# B&R Automation Studio project SD_SMA_SCADA_DEMO (part 2)

### Package Logical/SMA - SMA DataSQL demo

### GlobalDataSQL.typ - DataSQL types
```iecst
(*DataSQL types matching sma_data_collect OPC paths*)

TYPE
	DataSQLOperate_typ : 	STRUCT
		RecipeRead : BOOL;
		RecipeReadStatus : UINT;
		RecipeInsert : BOOL;
		RecipeInsertReq : BOOL;
		ProductRead : BOOL;
		ProductReadStatus : UINT;
		ProductInsert : BOOL;
		ProductInsertReq : BOOL;
		ProductInsertStatus : UDINT;
		AuditRead : BOOL;
		AuditReadStatus : UINT;
		AuditInsertFault : BOOL;
		AlarmRead : BOOL;
		AlarmReadStatus : UINT;
		AlarmInsertFault : BOOL;
		BatchInsert : BOOL;
		BatchInfoInsert : BOOL;
		RecipeCollectEnable : BOOL;
		ProductCollectEnable : BOOL;
		AlarmCollectEnable : BOOL;
		AuditCollectEnable : BOOL;
		BatchCollectEnable : BOOL;
		BatchInfoCollectEnable : BOOL;
	END_STRUCT;
END_TYPE

TYPE
	DataSQLQueryConfig_typ : 	STRUCT
		StartTime : ARRAY[0..DATA_SQL_QUERY_SIZE_MINUS]OF STRING[20];
		EndTime : ARRAY[0..DATA_SQL_QUERY_SIZE_MINUS]OF STRING[20];
		PointName : ARRAY[0..DATA_SQL_QUERY_SIZE_MINUS]OF STRING[20];
		AuxQuery : ARRAY[0..DATA_SQL_QUERY_SIZE_MINUS]OF STRING[80];
	END_STRUCT;
	DataSQLQueryCmd_typ : 	STRUCT
		Next : BOOL;
	END_STRUCT;
	DataSQLQuery_typ : 	STRUCT
		Config : DataSQLQueryConfig_typ;
		Cmd : DataSQLQueryCmd_typ;
	END_STRUCT;
END_TYPE

(*Recipe insert snapshot - scalar, for collector trigger read*)
TYPE
	DataSQLRecipe_typ : 	STRUCT
		TimeStamp : DATE_AND_TIME;
		State : UDINT;
		CH00 : REAL;
		CH01 : REAL;
		CH02 : REAL;
		CH03 : REAL;
		CH04 : REAL;
		CH05 : REAL;
		CH06 : REAL;
		CH07 : REAL;
		CH08 : REAL;
		CH09 : REAL;
		CH10 : REAL;
		CH11 : REAL;
		CH12 : REAL;
		CH13 : REAL;
		CH14 : REAL;
		CH15 : REAL;
		CH16 : REAL;
		CH17 : REAL;
		CH18 : REAL;
		CH19 : REAL;
		CH20 : REAL;
		CH21 : REAL;
		CH22 : REAL;
		CH23 : REAL;
		CH24 : REAL;
		CH25 : REAL;
	END_STRUCT;
END_TYPE

(*Product insert snapshot*)
TYPE
	DataSQLProduct_typ : 	STRUCT
		TimeStamp : DATE_AND_TIME;
		State : UDINT;
		CH01 : REAL;
		CH02 : REAL;
		CH03 : REAL;
		CH04 : REAL;
		CH05 : REAL;
		CH06 : REAL;
	END_STRUCT;
END_TYPE

TYPE
	DataSQLBatch_typ : 	STRUCT
		BatchCode : STRING[40];
		BatchTimeStart : DATE_AND_TIME;
		BatchTimeStop : DATE_AND_TIME;
	END_STRUCT;
END_TYPE

TYPE
	DataSQLBatchInfo_typ : 	STRUCT
		InfoProductName : STRING[80];
		InfoProductDesc : STRING[80];
		InfoConfigure : STRING[80];
		InfoRecipe : STRING[80];
		InfoTabletWeight : REAL;
		InfoTabletHardness : REAL;
		InfoTabletMoldXY : STRING[40];
		InfoTabletDiameterX : REAL;
		InfoTabletDiameterY : REAL;
		InfoTabletMoldZ : STRING[40];
		InfoTabletThicknessZ : REAL;
		InfoTabletRadiusR : REAL;
		InfoBatchStart : DATE_AND_TIME;
		InfoBatchStop : DATE_AND_TIME;
		InfoBatchRun : TIME;
		InfoPieceAccept : UDINT;
		InfoPieceDebug : UDINT;
		InfoPieceTotal : UDINT;
	END_STRUCT;
END_TYPE

(*Parallel Alarm insert buffer - all subscribed points are arrays*)
TYPE
	AlarmInsertBuffer_typ : 	STRUCT
		AlarmTime : ARRAY[0..DATA_SQL_PARALLEL_SIZE_MINUS]OF DATE_AND_TIME;
		AlarmCode : ARRAY[0..DATA_SQL_PARALLEL_SIZE_MINUS]OF UDINT;
		AlarmState : ARRAY[0..DATA_SQL_PARALLEL_SIZE_MINUS]OF UDINT;
		AlarmText : ARRAY[0..DATA_SQL_PARALLEL_SIZE_MINUS]OF STRING[80];
		InsertTrigger : ARRAY[0..DATA_SQL_PARALLEL_SIZE_MINUS]OF BOOL;
		AlarmBatch : ARRAY[0..DATA_SQL_PARALLEL_SIZE_MINUS]OF STRING[40];
	END_STRUCT;
END_TYPE

(*Parallel Audit insert buffer - all subscribed points are arrays*)
TYPE
	AuditInsertBuffer_typ : 	STRUCT
		AuditTime : ARRAY[0..DATA_SQL_PARALLEL_SIZE_MINUS]OF DATE_AND_TIME;
		AuditOperator : ARRAY[0..DATA_SQL_PARALLEL_SIZE_MINUS]OF STRING[32];
		AuditText : ARRAY[0..DATA_SQL_PARALLEL_SIZE_MINUS]OF STRING[100];
		InsertTrigger : ARRAY[0..DATA_SQL_PARALLEL_SIZE_MINUS]OF BOOL;
		AuditBatch : ARRAY[0..DATA_SQL_PARALLEL_SIZE_MINUS]OF STRING[40];
	END_STRUCT;
END_TYPE
```

### GlobalDataSQL.var - DataSQL globals
```iecst
(*DataSQL constants / globals matching sma_data_collect*)
VAR CONSTANT
	DATA_SQL_QUERY_SIZE : UINT := 30;
	DATA_SQL_QUERY_SIZE_MINUS : UINT := DATA_SQL_QUERY_SIZE - 1;
	(*Parallel Alarm/Audit buffer size (is_parallel)*)
	DATA_SQL_PARALLEL_SIZE : UINT := 100;
	DATA_SQL_PARALLEL_SIZE_MINUS : UINT := DATA_SQL_PARALLEL_SIZE - 1;
END_VAR
VAR
	gDataSQLHeartBeat : UINT;
	gDataSQLCommFault : BOOL;
	gDataSQLOperate : DataSQLOperate_typ;
	gDataSQLRecipe : DataSQLRecipe_typ;
	gDataSQLProduct : DataSQLProduct_typ;
	gDataSQLBatch : DataSQLBatch_typ;
	gDataSQLBatchInfo : DataSQLBatchInfo_typ;
	gDataSQLBatchOpen : BOOL;
END_VAR
```

### Program Logical/SMA/DataSQLAla (IEC) - Alarm insert buffer

#### Variables.var
```iecst
(*Alarm insert buffer + query - OPC ::DataSQLAla: (parallel arrays)*)
VAR
	AlarmInsertBuffer : AlarmInsertBuffer_typ;
	AlarmDataSQLQuery : DataSQLQuery_typ;
	UtcDTGetTime_0 : UtcDTGetTime;
	tonAlarm : TON;
	dtNow : DATE_AND_TIME;
	diAlarmCode : DINT;
	strTmp : STRING[16];
	usiIdx : USINT;
	bSimEnable : BOOL := TRUE;
	bManualTrigger : BOOL;
	uiManualIndex : UINT;
	iEvent : INT;
	iEventCount : INT;
	iIdx : INT;
END_VAR
```

#### Main.st
```iecst
PROGRAM _INIT
	AlarmDataSQLQuery.Config.PointName[0] := 'AlarmTime';
	AlarmDataSQLQuery.Config.PointName[1] := 'AlarmCode';
	AlarmDataSQLQuery.Config.PointName[2] := 'AlarmState';
	AlarmDataSQLQuery.Config.PointName[3] := 'AlarmText';
	bSimEnable := TRUE;
END_PROGRAM

PROGRAM _CYCLIC
	(*Fill AlarmInsertBuffer arrays (AlarmInsertBuffer_typ), then set InsertTrigger[i]*)
	UtcDTGetTime_0.enable := TRUE;
	UtcDTGetTime_0();
	IF UtcDTGetTime_0.status = 0 THEN
		dtNow := UtcDTGetTime_0.DT1;
	END_IF

	tonAlarm(IN := bSimEnable AND gDataSQLBatchOpen AND NOT tonAlarm.Q, PT := T#12s);

	IF tonAlarm.Q OR bManualTrigger THEN
		IF bManualTrigger THEN
			iEventCount := 1;
			iIdx := UINT_TO_INT(uiManualIndex MOD DATA_SQL_PARALLEL_SIZE);
			bManualTrigger := FALSE;
		ELSE
			iEventCount := DINT_TO_INT(RandRange(1, 3));
			iIdx := DINT_TO_INT(RandRange(0, 99));
		END_IF

		FOR iEvent := 0 TO iEventCount - 1 DO
			usiIdx := INT_TO_USINT((iIdx + (iEvent * 17)) MOD 100);
			IF NOT AlarmInsertBuffer.InsertTrigger[usiIdx] THEN
				diAlarmCode := RandRange(1000, 1049);
				AlarmInsertBuffer.AlarmTime[usiIdx] := dtNow;
				AlarmInsertBuffer.AlarmCode[usiIdx] := DINT_TO_UDINT(diAlarmCode);
				AlarmInsertBuffer.AlarmState[usiIdx] := DINT_TO_UDINT(RandRange(0, 1));
				strTmp := '';
				brsitoa(diAlarmCode, ADR(strTmp));
				AlarmInsertBuffer.AlarmText[usiIdx] := 'PRESS_FAULT_';
				brsstrcat(ADR(AlarmInsertBuffer.AlarmText[usiIdx]), ADR(strTmp));
				AlarmInsertBuffer.AlarmBatch[usiIdx] := gDataSQLBatch.BatchCode;
				AlarmInsertBuffer.InsertTrigger[usiIdx] := TRUE;
			END_IF
		END_FOR
	END_IF
END_PROGRAM

PROGRAM _EXIT

END_PROGRAM
```

### Program Logical/SMA/DataSQLAud (IEC) - Audit insert buffer

#### Variables.var
```iecst
(*Audit insert buffer + query - OPC ::DataSQLAud: (parallel arrays)*)
VAR
	AuditInsertBuffer : AuditInsertBuffer_typ;
	AuditDataSQLQuery : DataSQLQuery_typ;
	UtcDTGetTime_0 : UtcDTGetTime;
	tonAudit : TON;
	dtNow : DATE_AND_TIME;
	diAuditIdx : DINT;
	strTmp : STRING[16];
	usiIdx : USINT;
	bSimEnable : BOOL := TRUE;
	bManualTrigger : BOOL;
	uiManualIndex : UINT;
	iEvent : INT;
	iEventCount : INT;
	iIdx : INT;
END_VAR
```

#### Main.st
```iecst
PROGRAM _INIT
	AuditDataSQLQuery.Config.PointName[0] := 'AuditTime';
	AuditDataSQLQuery.Config.PointName[1] := 'AuditOperator';
	AuditDataSQLQuery.Config.PointName[2] := 'AuditText';
	bSimEnable := TRUE;
END_PROGRAM

PROGRAM _CYCLIC
	(*Fill AuditInsertBuffer arrays (AuditInsertBuffer_typ), then set InsertTrigger[i]*)
	UtcDTGetTime_0.enable := TRUE;
	UtcDTGetTime_0();
	IF UtcDTGetTime_0.status = 0 THEN
		dtNow := UtcDTGetTime_0.DT1;
	END_IF

	tonAudit(IN := bSimEnable AND gDataSQLBatchOpen AND NOT tonAudit.Q, PT := T#15s);

	IF tonAudit.Q OR bManualTrigger THEN
		IF bManualTrigger THEN
			iEventCount := 1;
			iIdx := UINT_TO_INT(uiManualIndex MOD DATA_SQL_PARALLEL_SIZE);
			bManualTrigger := FALSE;
		ELSE
			iEventCount := DINT_TO_INT(RandRange(1, 3));
			iIdx := DINT_TO_INT(RandRange(0, 99));
		END_IF

		FOR iEvent := 0 TO iEventCount - 1 DO
			usiIdx := INT_TO_USINT((iIdx + (iEvent * 23)) MOD 100);
			IF NOT AuditInsertBuffer.InsertTrigger[usiIdx] THEN
				diAuditIdx := RandRange(1, 12);
				strTmp := '';
				brsitoa(diAuditIdx, ADR(strTmp));
				AuditInsertBuffer.AuditTime[usiIdx] := dtNow;
				AuditInsertBuffer.AuditOperator[usiIdx] := 'Operator';
				brsstrcat(ADR(AuditInsertBuffer.AuditOperator[usiIdx]), ADR(strTmp));
				AuditInsertBuffer.AuditText[usiIdx] := 'PARAMETER_CHANGE_';
				brsstrcat(ADR(AuditInsertBuffer.AuditText[usiIdx]), ADR(strTmp));
				AuditInsertBuffer.AuditBatch[usiIdx] := gDataSQLBatch.BatchCode;
				AuditInsertBuffer.InsertTrigger[usiIdx] := TRUE;
			END_IF
		END_FOR
	END_IF
END_PROGRAM

PROGRAM _EXIT

END_PROGRAM
```

### Program Logical/SMA/DataSQLRec (IEC) - Recipe data + query

#### Variables.var
```iecst
(*Recipe query + random insert - OPC ::DataSQLRec: / ::AsGlobalPV:gDataSQLRecipe*)
VAR
	RecipeDataSQLQuery : DataSQLQuery_typ;
	UtcDTGetTime_0 : UtcDTGetTime;
	tonRecipe : TON;
	dtNow : DATE_AND_TIME;
	bSimEnable : BOOL := TRUE;
	bManualTrigger : BOOL;
	diRecipeProfile : DINT;
END_VAR
```

#### Main.st
```iecst
PROGRAM _INIT
	RecipeDataSQLQuery.Config.PointName[0] := 'DataRecipeTime';
	RecipeDataSQLQuery.Config.PointName[1] := 'DataRecipeState';
	RecipeDataSQLQuery.Config.PointName[2] := 'DataRecipeCH00';
	RecipeDataSQLQuery.Config.PointName[3] := 'DataRecipeCH01';
	RecipeDataSQLQuery.Config.PointName[4] := 'DataRecipeCH02';
	RecipeDataSQLQuery.Config.PointName[5] := 'DataRecipeCH03';
	RecipeDataSQLQuery.Config.PointName[6] := 'DataRecipeCH04';
	RecipeDataSQLQuery.Config.PointName[7] := 'DataRecipeCH05';
	RecipeDataSQLQuery.Config.PointName[8] := 'DataRecipeCH06';
	RecipeDataSQLQuery.Config.PointName[9] := 'DataRecipeCH07';
	RecipeDataSQLQuery.Config.PointName[10] := 'DataRecipeCH08';
	RecipeDataSQLQuery.Config.PointName[11] := 'DataRecipeCH09';
	RecipeDataSQLQuery.Config.PointName[12] := 'DataRecipeCH10';
	RecipeDataSQLQuery.Config.PointName[13] := 'DataRecipeCH11';
	RecipeDataSQLQuery.Config.PointName[14] := 'DataRecipeCH12';
	RecipeDataSQLQuery.Config.PointName[15] := 'DataRecipeCH13';
	RecipeDataSQLQuery.Config.PointName[16] := 'DataRecipeCH14';
	RecipeDataSQLQuery.Config.PointName[17] := 'DataRecipeCH15';
	RecipeDataSQLQuery.Config.PointName[18] := 'DataRecipeCH16';
	RecipeDataSQLQuery.Config.PointName[19] := 'DataRecipeCH17';
	RecipeDataSQLQuery.Config.PointName[20] := 'DataRecipeCH18';
	RecipeDataSQLQuery.Config.PointName[21] := 'DataRecipeCH19';
	RecipeDataSQLQuery.Config.PointName[22] := 'DataRecipeCH20';
	RecipeDataSQLQuery.Config.PointName[23] := 'DataRecipeCH21';
	RecipeDataSQLQuery.Config.PointName[24] := 'DataRecipeCH22';
	RecipeDataSQLQuery.Config.PointName[25] := 'DataRecipeCH23';
	RecipeDataSQLQuery.Config.PointName[26] := 'DataRecipeCH24';
	RecipeDataSQLQuery.Config.PointName[27] := 'DataRecipeCH25';
	bSimEnable := TRUE;
END_PROGRAM

PROGRAM _CYCLIC
	(*Fill gDataSQLRecipe (DataSQLRecipe_typ), then set RecipeInsert*)
	UtcDTGetTime_0.enable := TRUE;
	UtcDTGetTime_0();
	IF UtcDTGetTime_0.status = 0 THEN
		dtNow := UtcDTGetTime_0.DT1;
	END_IF

	(*Recipes change less frequently than product samples. PVI can request an extra snapshot.*)
	tonRecipe(IN := bSimEnable AND gDataSQLBatchOpen AND NOT gDataSQLOperate.RecipeInsert, PT := T#30s);
	IF EDGEPOS(tonRecipe.Q) OR EDGEPOS(gDataSQLBatchOpen) OR (bManualTrigger AND NOT gDataSQLOperate.RecipeInsert) THEN
		bManualTrigger := FALSE;
		diRecipeProfile := RandRange(1, 3);
		gDataSQLRecipe.TimeStamp := dtNow;
		gDataSQLRecipe.State := DINT_TO_UDINT(diRecipeProfile);
		CASE diRecipeProfile OF
			1:
				gDataSQLRecipe.CH00 := 0.500;
				gDataSQLRecipe.CH01 := 55.0;
				gDataSQLRecipe.CH02 := 9.00;
				gDataSQLRecipe.CH03 := 3.50;
				gDataSQLRecipe.CH04 := 72.0;
			2:
				gDataSQLRecipe.CH00 := 0.650;
				gDataSQLRecipe.CH01 := 62.0;
				gDataSQLRecipe.CH02 := 10.00;
				gDataSQLRecipe.CH03 := 4.00;
				gDataSQLRecipe.CH04 := 64.0;
			ELSE
				gDataSQLRecipe.CH00 := 0.350;
				gDataSQLRecipe.CH01 := 48.0;
				gDataSQLRecipe.CH02 := 8.00;
				gDataSQLRecipe.CH03 := 3.00;
				gDataSQLRecipe.CH04 := 80.0;
		END_CASE
		gDataSQLRecipe.CH05 := RandRangeReal(8.0, 12.0);
		gDataSQLRecipe.CH06 := RandRangeReal(18.0, 24.0);
		gDataSQLRecipe.CH07 := RandRangeReal(0.8, 1.2);
		gDataSQLRecipe.CH08 := RandRangeReal(2.0, 4.0);
		gDataSQLRecipe.CH09 := RandRangeReal(4.0, 7.0);
		gDataSQLRecipe.CH10 := RandRangeReal(35.0, 45.0);
		gDataSQLRecipe.CH11 := RandRangeReal(0.5, 1.0);
		gDataSQLRecipe.CH12 := RandRangeReal(0.5, 1.0);
		gDataSQLRecipe.CH13 := RandRangeReal(2.0, 4.0);
		gDataSQLRecipe.CH14 := RandRangeReal(10.0, 16.0);
		gDataSQLRecipe.CH15 := RandRangeReal(0.2, 0.8);
		gDataSQLRecipe.CH16 := RandRangeReal(0.2, 0.8);
		gDataSQLRecipe.CH17 := RandRangeReal(7.0, 10.0);
		gDataSQLRecipe.CH18 := RandRangeReal(7.0, 10.0);
		gDataSQLRecipe.CH19 := RandRangeReal(20.0, 30.0);
		gDataSQLRecipe.CH20 := RandRangeReal(20.0, 30.0);
		gDataSQLRecipe.CH21 := RandRangeReal(80.0, 120.0);
		gDataSQLRecipe.CH22 := RandRangeReal(80.0, 120.0);
		gDataSQLRecipe.CH23 := DINT_TO_REAL(diRecipeProfile);
		gDataSQLRecipe.CH24 := 100000.0;
		gDataSQLRecipe.CH25 := 1.0;
		gDataSQLOperate.RecipeInsert := TRUE;
	END_IF
END_PROGRAM

PROGRAM _EXIT

END_PROGRAM
```

### Program Logical/SMA/DataSQLPro (IEC) - Product data + query

#### Variables.var
```iecst
(*Product query + random insert - OPC ::DataSQLPro: / ::AsGlobalPV:gDataSQLProduct*)
VAR
	ProductDataSQLQuery : DataSQLQuery_typ;
	UtcDTGetTime_0 : UtcDTGetTime;
	tonProductData : TON;
	tonProductTrigger : TON;
	dtNow : DATE_AND_TIME;
	bSimEnable : BOOL := TRUE;
	bManualTrigger : BOOL;
	rProcessDrift : REAL;
END_VAR
```

#### Main.st
```iecst
PROGRAM _INIT
	ProductDataSQLQuery.Config.PointName[0] := 'DataProductTime';
	ProductDataSQLQuery.Config.PointName[1] := 'DataProductState';
	ProductDataSQLQuery.Config.PointName[2] := 'DataProductCH01';
	ProductDataSQLQuery.Config.PointName[3] := 'DataProductCH02';
	ProductDataSQLQuery.Config.PointName[4] := 'DataProductCH03';
	ProductDataSQLQuery.Config.PointName[5] := 'DataProductCH04';
	ProductDataSQLQuery.Config.PointName[6] := 'DataProductCH05';
	ProductDataSQLQuery.Config.PointName[7] := 'DataProductCH06';
	bSimEnable := TRUE;
END_PROGRAM

PROGRAM _CYCLIC
	(*Fill gDataSQLProduct (DataSQLProduct_typ), then set ProductInsert*)
	UtcDTGetTime_0.enable := TRUE;
	UtcDTGetTime_0();
	IF UtcDTGetTime_0.status = 0 THEN
		dtNow := UtcDTGetTime_0.DT1;
	END_IF

	(*Refresh process values every second so 5 s time collection sees changing data.*)
	tonProductData(IN := bSimEnable AND gDataSQLBatchOpen AND NOT tonProductData.Q, PT := T#1s);
	IF tonProductData.Q THEN
		rProcessDrift := rProcessDrift + RandRangeReal(-0.004, 0.004);
		IF rProcessDrift > 0.030 THEN
			rProcessDrift := 0.030;
		ELSIF rProcessDrift < -0.030 THEN
			rProcessDrift := -0.030;
		END_IF
		gDataSQLProduct.TimeStamp := dtNow;
		gDataSQLProduct.State := 2;
		gDataSQLProduct.CH01 := gDataSQLRecipe.CH00 + rProcessDrift + RandRangeReal(-0.010, 0.010);
		gDataSQLProduct.CH02 := gDataSQLRecipe.CH01 + RandRangeReal(-2.0, 2.0);
		gDataSQLProduct.CH03 := gDataSQLRecipe.CH03 + RandRangeReal(-0.08, 0.08);
		gDataSQLProduct.CH04 := gDataSQLRecipe.CH02 + RandRangeReal(-0.05, 0.05);
		gDataSQLProduct.CH05 := gDataSQLRecipe.CH05 + RandRangeReal(-0.5, 0.5);
		gDataSQLProduct.CH06 := gDataSQLRecipe.CH07 + RandRangeReal(-0.05, 0.05);
	END_IF

	(*Variable-trigger cadence is deliberately slower than the 5 s time trigger.*)
	tonProductTrigger(IN := bSimEnable AND gDataSQLBatchOpen AND NOT gDataSQLOperate.ProductInsert, PT := T#25s);
	IF EDGEPOS(tonProductTrigger.Q) OR (bManualTrigger AND NOT gDataSQLOperate.ProductInsert) THEN
		bManualTrigger := FALSE;
		gDataSQLProduct.TimeStamp := dtNow;
		gDataSQLOperate.ProductInsert := TRUE;
	END_IF
END_PROGRAM

PROGRAM _EXIT

END_PROGRAM
```

### Program Logical/SMA/DataSQLBat (IEC) - Batch / BatchInfo data

#### Main.st - Init, cyclic, exit code
```iecst
PROGRAM _INIT
	UtcDTGetTime_0.enable := TRUE;
	UtcDTGetTime_0();
	IF UtcDTGetTime_0.status = 0 THEN
		dtNow := UtcDTGetTime_0.DT1;
	END_IF

	diBatchSeq := DT_TO_DINT(dtNow);
	bSimEnable := TRUE;
	bBatchOpened := FALSE;
	gDataSQLBatchOpen := FALSE;

	(*No phantom open batch after startup. The first open is emitted after the idle timer.*)
	gDataSQLBatch.BatchCode := '';
	gDataSQLBatch.BatchTimeStart := DT#1970-01-01-00:00:00;
	gDataSQLBatch.BatchTimeStop := DT#1970-01-01-00:00:00;

	(*Initial gDataSQLBatchInfo (DataSQLBatchInfo_typ)*)
	gDataSQLBatchInfo.InfoProductName := 'SMA Tablet';
	gDataSQLBatchInfo.InfoProductDesc := 'Production simulation';
	gDataSQLBatchInfo.InfoConfigure := 'CFG_CP1586';
	gDataSQLBatchInfo.InfoRecipe := 'RCP_AUTO';
	gDataSQLBatchInfo.InfoTabletMoldXY := 'ROUND';
	gDataSQLBatchInfo.InfoTabletMoldZ := 'FLAT';
	gDataSQLBatchInfo.InfoBatchStart := dtNow;
	gDataSQLBatchInfo.InfoBatchStop := DT#1970-01-01-00:00:00;

	(*Collector groups are enabled by default; external OPC UA clients may toggle each flag.*)
	gDataSQLOperate.RecipeCollectEnable := TRUE;
	gDataSQLOperate.ProductCollectEnable := TRUE;
	gDataSQLOperate.AlarmCollectEnable := TRUE;
	gDataSQLOperate.AuditCollectEnable := TRUE;
	gDataSQLOperate.BatchCollectEnable := TRUE;
	gDataSQLOperate.BatchInfoCollectEnable := TRUE;
END_PROGRAM

PROGRAM _CYCLIC
	UtcDTGetTime_0.enable := TRUE;
	UtcDTGetTime_0();
	IF UtcDTGetTime_0.status = 0 THEN
		dtNow := UtcDTGetTime_0.DT1;
	END_IF

	(*Shared heartbeat for collector*)
	gDataSQLHeartBeat := gDataSQLHeartBeat + 1;

	(*Automatic cycle: 5 s changeover followed by 90 s production.*)
	tonBatchIdle(IN := bSimEnable AND NOT bBatchOpened AND NOT gDataSQLOperate.BatchInsert, PT := T#5s);
	tonBatchRun(IN := bSimEnable AND bBatchOpened AND NOT gDataSQLOperate.BatchInsert, PT := T#90s);
	IF tonBatchIdle.Q OR (uiManualCommand = 1 AND NOT bBatchOpened AND NOT gDataSQLOperate.BatchInsert) THEN
		uiManualCommand := 0;
		diBatchSeq := DT_TO_DINT(dtNow);
		IF diBatchSeq < 0 THEN
			diBatchSeq := -diBatchSeq;
		END_IF
			strTmp := '';
			brsitoa(diBatchSeq, ADR(strTmp));
			gDataSQLBatch.BatchCode := 'SMA_';
			brsstrcat(ADR(gDataSQLBatch.BatchCode), ADR(strTmp));
			gDataSQLBatch.BatchTimeStart := dtNow;
			gDataSQLBatch.BatchTimeStop := DT#1970-01-01-00:00:00;
			gDataSQLBatchInfo.InfoBatchStart := dtNow;
			gDataSQLBatchInfo.InfoBatchStop := DT#1970-01-01-00:00:00;
			gDataSQLBatchInfo.InfoPieceAccept := 0;
			gDataSQLBatchInfo.InfoPieceDebug := 0;
			gDataSQLBatchInfo.InfoPieceTotal := 0;
			bBatchOpened := TRUE;
			gDataSQLBatchOpen := TRUE;
		gDataSQLOperate.BatchInsert := TRUE;
	ELSIF tonBatchRun.Q OR (uiManualCommand = 2 AND bBatchOpened AND NOT gDataSQLOperate.BatchInsert) THEN
		uiManualCommand := 0;
		gDataSQLBatch.BatchTimeStop := dtNow;
		gDataSQLBatchInfo.InfoBatchStop := dtNow;
		gDataSQLBatchInfo.InfoBatchRun := dtNow - gDataSQLBatchInfo.InfoBatchStart;
		bBatchOpened := FALSE;
		gDataSQLBatchOpen := FALSE;
		gDataSQLOperate.BatchInsert := TRUE;
	END_IF

	(*Monotonic batch counters and measurements correlated with the active recipe.*)
	tonBatchInfo(IN := bSimEnable AND bBatchOpened AND NOT gDataSQLOperate.BatchInfoInsert, PT := T#10s);
	IF EDGEPOS(tonBatchInfo.Q) THEN
		gDataSQLBatchInfo.InfoProductName := 'SMA Tablet';
		gDataSQLBatchInfo.InfoProductDesc := 'Production simulation';
		gDataSQLBatchInfo.InfoConfigure := 'CFG_CP1586';
		gDataSQLBatchInfo.InfoRecipe := 'RCP_AUTO';
		gDataSQLBatchInfo.InfoTabletWeight := gDataSQLProduct.CH01;
		gDataSQLBatchInfo.InfoTabletHardness := gDataSQLProduct.CH02;
		gDataSQLBatchInfo.InfoTabletMoldXY := 'ROUND';
		gDataSQLBatchInfo.InfoTabletDiameterX := gDataSQLProduct.CH04;
		gDataSQLBatchInfo.InfoTabletDiameterY := gDataSQLProduct.CH04 + RandRangeReal(-0.03, 0.03);
		gDataSQLBatchInfo.InfoTabletMoldZ := 'FLAT';
		gDataSQLBatchInfo.InfoTabletThicknessZ := gDataSQLProduct.CH03;
		gDataSQLBatchInfo.InfoTabletRadiusR := gDataSQLProduct.CH04 / 2.0;
		gDataSQLBatchInfo.InfoPieceAccept := gDataSQLBatchInfo.InfoPieceAccept + DINT_TO_UDINT(RandRange(80, 120));
		gDataSQLBatchInfo.InfoPieceDebug := gDataSQLBatchInfo.InfoPieceDebug + DINT_TO_UDINT(RandRange(0, 3));
		gDataSQLBatchInfo.InfoPieceTotal := gDataSQLBatchInfo.InfoPieceAccept + gDataSQLBatchInfo.InfoPieceDebug;
		IF bBatchOpened THEN
			gDataSQLBatchInfo.InfoBatchRun := dtNow - gDataSQLBatchInfo.InfoBatchStart;
		END_IF
		gDataSQLOperate.BatchInfoInsert := TRUE;
	END_IF
END_PROGRAM

PROGRAM _EXIT

END_PROGRAM
```

#### Variables.var - Local variables
```iecst
(*Batch / BatchInfo random insert - OPC ::AsGlobalPV:gDataSQLBatch / gDataSQLBatchInfo*)
VAR
	UtcDTGetTime_0 : UtcDTGetTime;
	tonBatchRun : TON;
	tonBatchIdle : TON;
	tonBatchInfo : TON;
	dtNow : DATE_AND_TIME;
	diBatchSeq : DINT;
	strTmp : STRING[16];
	bBatchOpened : BOOL;
	bSimEnable : BOOL := TRUE;
	uiManualCommand : UINT;
END_VAR
```

### Program Logical/SMA/LoadControl (IEC) - Closed-loop CPU load controller

#### Main.st - CPU load controller
```iecst
PROGRAM _INIT
	bEnable := TRUE;
	uiTargetLoadPercent := 50;

	fbRuntimeInfo.enable := TRUE;
	fbRuntimeInfo();
	udCycleTimeUs := fbRuntimeInfo.cycle_time;
	IF udCycleTimeUs = 0 THEN
		(* Cyclic #4 is normally 100 ms; this fallback is only used if RTInfo fails. *)
		udCycleTimeUs := 100000;
	END_IF

	(* Start below the target; the feedback loop converges without an initial spike. *)
	udBusyBudgetUs := udCycleTimeUs / 5;

	fbIdleMeasure.enable := TRUE;
	fbIdleMeasure.measurementPeriod := 500;
	fbIdleMeasure.measurementLevel := 1;
	fbIdleMeasure();
END_PROGRAM

PROGRAM _CYCLIC
	(* Read the configured task-class period instead of relying on a fixed cycle time. *)
	fbRuntimeInfo.enable := TRUE;
	fbRuntimeInfo();
	IF (fbRuntimeInfo.status = 0) AND (fbRuntimeInfo.cycle_time > 0) THEN
		udCycleTimeUs := fbRuntimeInfo.cycle_time;
	END_IF

	(* Keep the operator setpoint in a range that leaves watchdog headroom. *)
	IF uiTargetLoadPercent < 5 THEN
		uiTargetLoadPercent := 5;
	ELSIF uiTargetLoadPercent > 75 THEN
		uiTargetLoadPercent := 75;
	END_IF

	(* Idle rate is averaged by Automation Runtime over a 500 ms interval. *)
	fbIdleMeasure.enable := TRUE;
	fbIdleMeasure.measurementPeriod := 500;
	fbIdleMeasure.measurementLevel := 1;
	fbIdleMeasure();
	uiIdleStatus := fbIdleMeasure.status;
	IF (uiIdleStatus = 0) AND (fbIdleMeasure.idleRate <= 100) THEN
		udMeasuredLoadPercent := 100 - fbIdleMeasure.idleRate;
	END_IF

	(* Update once per measurement interval. Gain 0.5 avoids oscillation. *)
	udControlElapsedUs := udControlElapsedUs + udCycleTimeUs;
	IF udControlElapsedUs >= 500000 THEN
		udControlElapsedUs := udControlElapsedUs - 500000;

		IF bEnable AND (uiIdleStatus = 0) THEN
			diLoadError := UINT_TO_DINT(uiTargetLoadPercent) - UDINT_TO_DINT(udMeasuredLoadPercent);
			diCorrectionUs := (diLoadError * UDINT_TO_DINT(udCycleTimeUs)) / 200;
			diNewBudgetUs := UDINT_TO_DINT(udBusyBudgetUs) + diCorrectionUs;
			udMaxBudgetUs := (udCycleTimeUs * 75) / 100;

			IF diNewBudgetUs < 0 THEN
				udBusyBudgetUs := 0;
			ELSIF DINT_TO_UDINT(diNewBudgetUs) > udMaxBudgetUs THEN
				udBusyBudgetUs := udMaxBudgetUs;
			ELSE
				udBusyBudgetUs := DINT_TO_UDINT(diNewBudgetUs);
			END_IF
		ELSIF NOT bEnable THEN
			udBusyBudgetUs := 0;
		END_IF
	END_IF

	IF bEnable AND (udBusyBudgetUs > 0) THEN
		(* Build a microsecond timestamp within the current second.  Re-read the
		   tick if it rolled while TIM_musec() was sampled. *)
		uiTick := TIM_ticks();
		uiMicrosecond := TIM_musec();
		uiTickCheck := TIM_ticks();
		IF uiTickCheck <> uiTick THEN
			uiTick := uiTickCheck;
			uiMicrosecond := TIM_musec();
		END_IF
		udStartUs := UINT_TO_UDINT(uiTick) * 10000 + UINT_TO_UDINT(uiMicrosecond);
		udElapsedUs := 0;

		WHILE udElapsedUs < udBusyBudgetUs DO
			uiTick := TIM_ticks();
			uiMicrosecond := TIM_musec();
			uiTickCheck := TIM_ticks();
			IF uiTickCheck <> uiTick THEN
				uiTick := uiTickCheck;
				uiMicrosecond := TIM_musec();
			END_IF
			udNowUs := UINT_TO_UDINT(uiTick) * 10000 + UINT_TO_UDINT(uiMicrosecond);

			IF udNowUs >= udStartUs THEN
				udElapsedUs := udNowUs - udStartUs;
			ELSE
				(* TIM_ticks() wraps every second. *)
				udElapsedUs := (1000000 - udStartUs) + udNowUs;
			END_IF
		END_WHILE
	END_IF
END_PROGRAM

PROGRAM _EXIT
	fbIdleMeasure.enable := FALSE;
	fbIdleMeasure();
END_PROGRAM
```

#### Variables.var - Controller variables
```iecst
VAR
	(* Online controls and diagnostics. *)
	bEnable : BOOL := TRUE;
	uiTargetLoadPercent : UINT := 50;
	udMeasuredLoadPercent : UDINT;
	udBusyBudgetUs : UDINT;
	udCycleTimeUs : UDINT;
	uiIdleStatus : UINT;

	(* Internal controller state. *)
	fbIdleMeasure : LogIdleShow;
	fbRuntimeInfo : RTInfo;
	udControlElapsedUs : UDINT;
	diLoadError : DINT;
	diCorrectionUs : DINT;
	diNewBudgetUs : DINT;
	udMaxBudgetUs : UDINT;
	udStartUs : UDINT;
	udNowUs : UDINT;
	udElapsedUs : UDINT;
	uiTick : UINT;
	uiTickCheck : UINT;
	uiMicrosecond : UINT;
END_VAR
```

### GlobalDataSQL.typ - not listed in the package file held
```iecst
(*DataSQL types matching sma_data_collect OPC paths*)

TYPE
	DataSQLOperate_typ : 	STRUCT
		RecipeRead : BOOL;
		RecipeReadStatus : UINT;
		RecipeInsert : BOOL;
		RecipeInsertReq : BOOL;
		ProductRead : BOOL;
		ProductReadStatus : UINT;
		ProductInsert : BOOL;
		ProductInsertReq : BOOL;
		ProductInsertStatus : UDINT;
		AuditRead : BOOL;
		AuditReadStatus : UINT;
		AuditInsertFault : BOOL;
		AlarmRead : BOOL;
		AlarmReadStatus : UINT;
		AlarmInsertFault : BOOL;
		BatchInsert : BOOL;
		BatchInfoInsert : BOOL;
	END_STRUCT;
END_TYPE

TYPE
	DataSQLQueryConfig_typ : 	STRUCT
		StartTime : ARRAY[0..DATA_SQL_QUERY_SIZE_MINUS]OF STRING[20];
		EndTime : ARRAY[0..DATA_SQL_QUERY_SIZE_MINUS]OF STRING[20];
		PointName : ARRAY[0..DATA_SQL_QUERY_SIZE_MINUS]OF STRING[20];
		AuxQuery : ARRAY[0..DATA_SQL_QUERY_SIZE_MINUS]OF STRING[80];
	END_STRUCT;
	DataSQLQueryCmd_typ : 	STRUCT
		Next : BOOL;
	END_STRUCT;
	DataSQLQuery_typ : 	STRUCT
		Config : DataSQLQueryConfig_typ;
		Cmd : DataSQLQueryCmd_typ;
	END_STRUCT;
END_TYPE

(*Recipe insert snapshot - scalar, for collector trigger read*)
TYPE
	DataSQLRecipe_typ : 	STRUCT
		TimeStamp : DATE_AND_TIME;
		State : UDINT;
		CH00 : REAL;
		CH01 : REAL;
		CH02 : REAL;
		CH03 : REAL;
		CH04 : REAL;
		CH05 : REAL;
		CH06 : REAL;
		CH07 : REAL;
		CH08 : REAL;
		CH09 : REAL;
		CH10 : REAL;
		CH11 : REAL;
		CH12 : REAL;
		CH13 : REAL;
		CH14 : REAL;
		CH15 : REAL;
		CH16 : REAL;
		CH17 : REAL;
		CH18 : REAL;
		CH19 : REAL;
		CH20 : REAL;
		CH21 : REAL;
		CH22 : REAL;
		CH23 : REAL;
		CH24 : REAL;
		CH25 : REAL;
	END_STRUCT;
END_TYPE

(*Product insert snapshot*)
TYPE
	DataSQLProduct_typ : 	STRUCT
		TimeStamp : DATE_AND_TIME;
		State : UDINT;
		CH01 : REAL;
		CH02 : REAL;
		CH03 : REAL;
		CH04 : REAL;
		CH05 : REAL;
		CH06 : REAL;
	END_STRUCT;
END_TYPE

TYPE
	DataSQLBatch_typ : 	STRUCT
		BatchCode : STRING[40];
		BatchTimeStart : DATE_AND_TIME;
		BatchTimeStop : DATE_AND_TIME;
	END_STRUCT;
END_TYPE

TYPE
	DataSQLBatchInfo_typ : 	STRUCT
		InfoProductName : STRING[80];
		InfoProductDesc : STRING[80];
		InfoConfigure : STRING[80];
		InfoRecipe : STRING[80];
		InfoTabletWeight : REAL;
		InfoTabletHardness : REAL;
		InfoTabletMoldXY : STRING[40];
		InfoTabletDiameterX : REAL;
		InfoTabletDiameterY : REAL;
		InfoTabletMoldZ : STRING[40];
		InfoTabletThicknessZ : REAL;
		InfoTabletRadiusR : REAL;
		InfoBatchStart : DATE_AND_TIME;
		InfoBatchStop : DATE_AND_TIME;
		InfoBatchRun : TIME;
		InfoPieceAccept : UDINT;
		InfoPieceDebug : UDINT;
		InfoPieceTotal : UDINT;
	END_STRUCT;
END_TYPE

TYPE
	AlarmInsertBuffer_typ : 	STRUCT
		AlarmTime : DATE_AND_TIME;
		AlarmCode : UDINT;
		AlarmState : UDINT;
		AlarmText : STRING[80];
		InsertTrigger : BOOL;
		AlarmBatch : STRING[40];
	END_STRUCT;
END_TYPE

TYPE
	AuditInsertBuffer_typ : 	STRUCT
		AuditTime : DATE_AND_TIME;
		AuditOperator : STRING[32];
		AuditText : STRING[100];
		InsertTrigger : BOOL;
		AuditBatch : STRING[40];
	END_STRUCT;
END_TYPE
```

### GlobalDataSQL.var - not listed in the package file held
```iecst
(*DataSQL constants / globals matching sma_data_collect*)
VAR CONSTANT
	DATA_SQL_QUERY_SIZE : UINT := 30;
	DATA_SQL_QUERY_SIZE_MINUS : UINT := DATA_SQL_QUERY_SIZE - 1;
END_VAR
VAR
	gDataSQLHeartBeat : UINT;
	gDataSQLCommFault : BOOL;
	gDataSQLOperate : DataSQLOperate_typ;
	gDataSQLRecipe : DataSQLRecipe_typ;
	gDataSQLProduct : DataSQLProduct_typ;
	gDataSQLBatch : DataSQLBatch_typ;
	gDataSQLBatchInfo : DataSQLBatchInfo_typ;
END_VAR
```

### Program Logical/AlarmQuerry (IEC)

#### Main.st - Init, cyclic, exit code
```iecst
PROGRAM _INIT
	(* Insert code here *)
	stDbReadQuery.stConfig.strPointName[0] := 'msg';
	guiDBHeartBeat;

END_PROGRAM

PROGRAM _CYCLIC
	(* Insert code here *)
	//Data GEN - Alarm Group 1 Data Points
	// GET TIME
	UtcDTGetTime_0.enable := TRUE;
	UtcDTGetTime_0();
	IF UtcDTGetTime_0.status = 0 THEN
		ts := DT_TO_STRING(UtcDTGetTime_0.DT1);
	END_IF
	Code := RandRange(1,10);  // 报警码
	msg := RandRange(1,10);  // 报警信息
	severity := RandRange(1,4);  // 报警等级 (1=Critical, 2=Major, 3=Minor, 4=Info)
	Status := btrigger;  // 报警状态 (TRUE=Active, FALSE=Cleared)
	Batch ;  // 生产批号

	//Triggerrecord
	btrigger;

	//Data from DATABASE
	bExecuteRead;
	stDbReadQuery;

	//Para and button connect
	stDbReadQuery.stConfig.strStartTime[0] := '';
	brsstrcat(ADR(stDbReadQuery.stConfig.strStartTime[0]),ADR(HMIAlarmQuerrystYear));
	brsstrcat(ADR(stDbReadQuery.stConfig.strStartTime[0]),ADR('-'));
	brsstrcat(ADR(stDbReadQuery.stConfig.strStartTime[0]),ADR(HMIAlarmQuerrystMonth));
	brsstrcat(ADR(stDbReadQuery.stConfig.strStartTime[0]),ADR('-'));
	brsstrcat(ADR(stDbReadQuery.stConfig.strStartTime[0]),ADR(HMIAlarmQuerrystDay));
	brsstrcat(ADR(stDbReadQuery.stConfig.strStartTime[0]),ADR(' '));

	brsstrcat(ADR(stDbReadQuery.stConfig.strStartTime[0]),ADR(HMIAlarmQuerrystHour));
	brsstrcat(ADR(stDbReadQuery.stConfig.strStartTime[0]),ADR(':'));
	brsstrcat(ADR(stDbReadQuery.stConfig.strStartTime[0]),ADR(HMIAlarmQuerrystMinute));
	brsstrcat(ADR(stDbReadQuery.stConfig.strStartTime[0]),ADR(':'));
	brsstrcat(ADR(stDbReadQuery.stConfig.strStartTime[0]),ADR(HMIAlarmQuerrystSec));

	stDbReadQuery.stConfig.strEndTime[0] := '';
	brsstrcat(ADR(stDbReadQuery.stConfig.strEndTime[0]),ADR(HMIAlarmQuerryedYear));
	brsstrcat(ADR(stDbReadQuery.stConfig.strEndTime[0]),ADR('-'));
	brsstrcat(ADR(stDbReadQuery.stConfig.strEndTime[0]),ADR(HMIAlarmQuerryedMonth));
	brsstrcat(ADR(stDbReadQuery.stConfig.strEndTime[0]),ADR('-'));
	brsstrcat(ADR(stDbReadQuery.stConfig.strEndTime[0]),ADR(HMIAlarmQuerryedDay));
	brsstrcat(ADR(stDbReadQuery.stConfig.strEndTime[0]),ADR(' '));

	brsstrcat(ADR(stDbReadQuery.stConfig.strEndTime[0]),ADR(HMIAlarmQuerryedHour));
	brsstrcat(ADR(stDbReadQuery.stConfig.strEndTime[0]),ADR(':'));
	brsstrcat(ADR(stDbReadQuery.stConfig.strEndTime[0]),ADR(HMIAlarmQuerryedMinute));
	brsstrcat(ADR(stDbReadQuery.stConfig.strEndTime[0]),ADR(':'));
	brsstrcat(ADR(stDbReadQuery.stConfig.strEndTime[0]),ADR(HMIAlarmQuerryedSec));

	bExecuteRead := UINT_TO_BOOL(HMIAlarmQuerryMBBtn);

	//Response data
	FOR i := 0 TO MAX_ENTRIES_PERPAGE_MINUSONE DO
		IF stDbReadQuery.stRev[0].udiRevTime[i] <> 0 THEN
			//强制转换
			DT_TO_DTStructure(UDINT_TO_DT(stDbReadQuery.stRev[0].udiRevTime[i]),ADR(stRecvDT[i]));

			HMIAlarmQuerryTimestr[i] := '';

			brsitoa(UINT_TO_DINT(stRecvDT[i].year),ADR(strempYear));
			brsitoa(UINT_TO_DINT(stRecvDT[i].month),ADR(strempMonth));
			brsitoa(UINT_TO_DINT(stRecvDT[i].day),ADR(strempDay));
			brsitoa(UINT_TO_DINT(stRecvDT[i].hour),ADR(strempHour));
			brsitoa(UINT_TO_DINT(stRecvDT[i].minute),ADR(strempMinute));
			brsitoa(UINT_TO_DINT(stRecvDT[i].second),ADR(strtempSecond));

			brsstrcat(ADR(HMIAlarmQuerryTimestr[i]),ADR(strempYear));
			brsstrcat(ADR(HMIAlarmQuerryTimestr[i]),ADR('-'));
			brsstrcat(ADR(HMIAlarmQuerryTimestr[i]),ADR(strempMonth));
			brsstrcat(ADR(HMIAlarmQuerryTimestr[i]),ADR('-'));
			brsstrcat(ADR(HMIAlarmQuerryTimestr[i]),ADR(strempDay));
			brsstrcat(ADR(HMIAlarmQuerryTimestr[i]),ADR(' '));
			brsstrcat(ADR(HMIAlarmQuerryTimestr[i]),ADR(strempHour));
			brsstrcat(ADR(HMIAlarmQuerryTimestr[i]),ADR(':'));
			brsstrcat(ADR(HMIAlarmQuerryTimestr[i]),ADR(strempMinute));
			brsstrcat(ADR(HMIAlarmQuerryTimestr[i]),ADR(':'));
			brsstrcat(ADR(HMIAlarmQuerryTimestr[i]),ADR(strtempSecond));

		ELSE
			brsmemset(ADR(HMIAlarmQuerryTimestr[i]),0,SIZEOF(HMIAlarmQuerryTimestr[i]));
		END_IF
		HMIAlarmQuerryIndex[i] :=  REAL_TO_UINT(stDbReadQuery.stRev[0].rRevBuffer[i]);

	END_FOR

END_PROGRAM

PROGRAM _EXIT
	(* Insert code here *)

END_PROGRAM
```

#### Types.typ - Local data types
```iecst
(*DBQuery*)

TYPE
	dbReadConfig_typ : 	STRUCT
		strStartTime : ARRAY[0..DB_READ_QUERY_SIZE_MINUS_ONE]OF STRING[20];
		strEndTime : ARRAY[0..DB_READ_QUERY_SIZE_MINUS_ONE]OF STRING[20];
		strPointName : ARRAY[0..DB_READ_QUERY_SIZE_MINUS_ONE]OF STRING[20];
	END_STRUCT;
	dbReadRev_typ : 	STRUCT
		rRevBuffer : ARRAY[0..REV_BUFFER_SIZE_MINUS_ONE]OF REAL;
		udiRevTime : ARRAY[0..REV_BUFFER_SIZE_MINUS_ONE]OF UDINT;
	END_STRUCT;
	dbReadQuery_typ : 	STRUCT
		stConfig : dbReadConfig_typ;
		stRev : ARRAY[0..DB_READ_QUERY_SIZE_MINUS_ONE]OF dbReadRev_typ;
	END_STRUCT;
END_TYPE
```

#### Variables.var - Local variables
```iecst
(*HMIConnect*)
VAR
	HMIAlarmQuerrystYear : STRING[10];
	HMIAlarmQuerrystMonth : STRING[10];
	HMIAlarmQuerrystDay : STRING[10];
	HMIAlarmQuerrystHour : STRING[10];
	HMIAlarmQuerrystMinute : STRING[10];
	HMIAlarmQuerrystSec : STRING[10];
	HMIAlarmQuerryedYear : STRING[10];
	HMIAlarmQuerryedMonth : STRING[10];
	HMIAlarmQuerryedDay : STRING[10];
	HMIAlarmQuerryedHour : STRING[10];
	HMIAlarmQuerryedMinute : STRING[10];
	HMIAlarmQuerryedSec : STRING[10];
	HMIAlarmClearMBBtn : UINT;
	HMIAlarmQuerryMBBtn : UINT;
	HMIAlarmQuerryTimestr : ARRAY[0..MAX_ENTRIES_PERPAGE_MINUSONE] OF STRING[100];
	HMIAlarmQuerryIndex : ARRAY[0..MAX_ENTRIES_PERPAGE_MINUSONE] OF UINT;
END_VAR
(*DATA BASE Query*)
VAR
	bExecuteRead : BOOL;
	stDbReadQuery : dbReadQuery_typ;
END_VAR
(*DATA BASE CONSTANT*)
VAR CONSTANT
	REV_BUFFER_SIZE : UINT := 10000;
	REV_BUFFER_SIZE_MINUS_ONE : UINT := REV_BUFFER_SIZE-1;
	DB_READ_QUERY_SIZE : UINT := 10;
	DB_READ_QUERY_SIZE_MINUS_ONE : UINT := DB_READ_QUERY_SIZE-1;
END_VAR
(*Data point*)
VAR
	ts : STRING[80];
	Code : DINT;
	msg : DINT;
	Batch : DINT;
	severity : DINT;
	Status : DINT;
END_VAR
(*TIME CONVENT*)
VAR
	UtcDTGetTime_0 : UtcDTGetTime;
END_VAR
(*connect var*)
VAR
	stRecvDT : {REDUND_UNREPLICABLE} ARRAY[0..MAX_ENTRIES_PERPAGE_MINUSONE] OF DTStructure;
	strtempSecond : STRING[10];
	strempMinute : STRING[10];
	strempHour : STRING[10];
	strempDay : STRING[10];
	strempMonth : STRING[10];
	strempYear : STRING[10];
	i : UINT;
END_VAR
(*Insert your comment here.*)
VAR CONSTANT
	MAX_ENTRIES_PERPAGE_MINUSONE : UINT := MAX_ENTRIES_PERPAGE- 1;
	MAX_ENTRIES_PERPAGE : UINT := 15;
END_VAR
VAR
	btrigger : BOOL;
END_VAR
```

### Program Logical/DataGen

#### Variables.var
```iecst
VAR
	IP1 : DINT;
	IP2 : DINT;
	FP2 : REAL;
END_VAR
(*Insert your comment here.*)
VAR
	dtTimeStamp : DATE_AND_TIME;
	strTimeStamp : STRING[80];
	ID : DINT;
	STATE : DINT;
	TimeStamp : STRING[32];
	Millsec : DINT;
	CV : REAL;
	VPF : REAL;
	WT : REAL;
	F1 : REAL;
	F2 : REAL;
	F3 : REAL;
	F4 : REAL;
	F5 : REAL;
	F6 : REAL;
	F7 : REAL;
	F8 : REAL;
	F9 : REAL;
	F10 : REAL;
	F11 : REAL;
	F12 : REAL;
	F13 : REAL;
	F14 : REAL;
	F15 : REAL;
	FP : REAL;
	AP1 : REAL;
	BP1 : REAL;
	AP2 : REAL;
	ST1 : REAL;
	ST2 : REAL;
	ST3 : REAL;
	ST4 : REAL;
	ST5 : REAL;
	ST6 : REAL;
	ST7 : REAL;
	ST8 : REAL;
	ST9 : REAL;
	ST10 : REAL;
	ST11 : REAL;
	ST12 : REAL;
	ST13 : REAL;
	ST14 : REAL;
	ST15 : REAL;
	AIR : REAL;
	CP : REAL;
	CT : REAL;
	CRT : REAL;
	ES : REAL;
	FP1 : REAL;
	FT : REAL;
	FF : REAL;
	FC : DINT;
	HT1 : REAL;
	HT2 : REAL;
	HT3 : REAL;
	HT4 : REAL;
	HT5 : REAL;
	HT6 : REAL;
	HT7 : REAL;
	HT8 : REAL;
	HT9 : REAL;
	HT10 : REAL;
	HT11 : REAL;
	HT12 : REAL;
	HT13 : REAL;
	HT14 : REAL;
	HT15 : REAL;
	HT16 : REAL;
	HT17 : REAL;
	HT18 : REAL;
	HT19 : REAL;
	HT20 : REAL;
	MP : REAL;
	MT : REAL;
	MCT : REAL;
	MCP : REAL;
	EC : REAL;
	EST : REAL;
	ES1 : REAL;
	TC : REAL;
	TF : REAL;
	TW : REAL;
END_VAR
```

#### Main.st
```iecst
PROGRAM _INIT
	(* Insert code here *)

END_PROGRAM

PROGRAM _CYCLIC
	(* Insert code here *)
	strTimeStamp;
	strTimeStamp := DT_TO_STRING(dtTimeStamp);
	IP1 := RandINT();
	IP2 := RandINT();

	FP1 := RandRangeReal(0, 100);
	FP2 := RandRangeReal(0, 100);

	CV := RandRangeReal(0, 100);
	VPF := RandRangeReal(0, 100);
	WT := RandRangeReal(0, 100);

	F1 := RandRangeReal(0, 100);
	F2 := RandRangeReal(0, 100);
	F3 := RandRangeReal(0, 100);
	F4 := RandRangeReal(0, 100);
	F5 := RandRangeReal(0, 100);
	F6 := RandRangeReal(0, 100);
	F7 := RandRangeReal(0, 100);
	F8 := RandRangeReal(0, 100);
	F9 := RandRangeReal(0, 100);
	F10 := RandRangeReal(0, 100);
	F11 := RandRangeReal(0, 100);
	F12 := RandRangeReal(0, 100);
	F13 := RandRangeReal(0, 100);
	F14 := RandRangeReal(0, 100);
	F15 := RandRangeReal(0, 100);

	FP := RandRangeReal(0, 100);

	AP1 := RandRangeReal(0, 100);
	BP1 := RandRangeReal(0, 100);
	AP2 := RandRangeReal(0, 100);

	ST1 := RandRangeReal(0, 100);
	ST2 := RandRangeReal(0, 100);
	ST3 := RandRangeReal(0, 100);
	ST4 := RandRangeReal(0, 100);
	ST5 := RandRangeReal(0, 100);
	ST6 := RandRangeReal(0, 100);
	ST7 := RandRangeReal(0, 100);
	ST8 := RandRangeReal(0, 100);
	ST9 := RandRangeReal(0, 100);
	ST10 := RandRangeReal(0, 100);
	ST11 := RandRangeReal(0, 100);
	ST12 := RandRangeReal(0, 100);
	ST13 := RandRangeReal(0, 100);
	ST14 := RandRangeReal(0, 100);
	ST15 := RandRangeReal(0, 100);

	AIR := RandRangeReal(0, 100);
	CP := RandRangeReal(0, 100);
	CT := RandRangeReal(0, 100);
	CRT := RandRangeReal(0, 100);
	ES := RandRangeReal(0, 100);
	FT := RandRangeReal(0, 100);
	FF := RandRangeReal(0, 100);

	FC := RandINT();

	HT1 := RandRangeReal(0, 100);
	HT2 := RandRangeReal(0, 100);
	HT3 := RandRangeReal(0, 100);
	HT4 := RandRangeReal(0, 100);
	HT5 := RandRangeReal(0, 100);
	HT6 := RandRangeReal(0, 100);
	HT7 := RandRangeReal(0, 100);
	HT8 := RandRangeReal(0, 100);
	HT9 := RandRangeReal(0, 100);
	HT10 := RandRangeReal(0, 100);
	HT11 := RandRangeReal(0, 100);
	HT12 := RandRangeReal(0, 100);
	HT13 := RandRangeReal(0, 100);
	HT14 := RandRangeReal(0, 100);
	HT15 := RandRangeReal(0, 100);
	HT16 := RandRangeReal(0, 100);
	HT17 := RandRangeReal(0, 100);
	HT18 := RandRangeReal(0, 100);
	HT19 := RandRangeReal(0, 100);
	HT20 := RandRangeReal(0, 100);

	MP := RandRangeReal(0, 100);
	MT := RandRangeReal(0, 100);
	MCT := RandRangeReal(0, 100);
	MCP := RandRangeReal(0, 100);
	EC := RandRangeReal(0, 100);
	EST := RandRangeReal(0, 100);
	ES1 := RandRangeReal(0, 100);
	TC := RandRangeReal(0, 100);
	TF := RandRangeReal(0, 100);
	TW := RandRangeReal(0, 100);
END_PROGRAM

PROGRAM _EXIT
	(* Insert code here *)

END_PROGRAM
```

### Program Logical/DataRev

#### Types.typ
```iecst
TYPE
	dbReadConfig_typ : 	STRUCT
		strStartTime : ARRAY[0..DB_READ_QUERY_SIZE_MINUS_ONE]OF STRING[20];
		strEndTime : ARRAY[0..DB_READ_QUERY_SIZE_MINUS_ONE]OF STRING[20];
		strPointName : ARRAY[0..DB_READ_QUERY_SIZE_MINUS_ONE]OF STRING[20];
	END_STRUCT;
	dbReadRev_typ : 	STRUCT
		rRevBuffer : ARRAY[0..REV_BUFFER_SIZE_MINUS_ONE]OF REAL;
		udiRevTime : ARRAY[0..REV_BUFFER_SIZE_MINUS_ONE]OF UDINT;
		udiRevFeedBack : UDINT;
	END_STRUCT;
	dbReadQuery_typ : 	STRUCT
		stConfig : dbReadConfig_typ;
		stCmd : dbReadCmd_typ;
		stRev : ARRAY[0..DB_READ_QUERY_SIZE_MINUS_ONE]OF dbReadRev_typ;
	END_STRUCT;
	dbReadCmd_typ : 	STRUCT
		bNext : BOOL;
	END_STRUCT;
END_TYPE
```

#### Variables.var
```iecst
(*Insert your comment here.*)
VAR
	bExecuteRead : BOOL;
	stDbReadQuery : dbReadQuery_typ;
	bTestTriger : BOOL;
	uiHeartBeat : UINT;
	uiQueryFeedBack : UINT;
END_VAR
```

#### Main.st
```iecst
PROGRAM _INIT
	(* Insert code here *)
	// 同一次查询，目前最好设定查询时间一致
	stDbReadQuery.stConfig.strPointName[0] := 'rAP1';
	stDbReadQuery.stConfig.strStartTime[0] := '2026-03-04 15:21:32';
	stDbReadQuery.stConfig.strEndTime[0]   := '2026-03-05 15:21:32';

	stDbReadQuery.stConfig.strPointName[1] := 'rF10';
	stDbReadQuery.stConfig.strStartTime[1] := '2026-03-04 15:21:32';
	stDbReadQuery.stConfig.strEndTime[1]   := '2026-03-04 15:21:32';

	stDbReadQuery.stConfig.strPointName[1] := 'rF11';
	stDbReadQuery.stConfig.strStartTime[1] := '2026-03-04 15:21:32';
	stDbReadQuery.stConfig.strEndTime[1]   := '2026-03-04 15:21:32';

	stDbReadQuery.stConfig.strPointName[1] := 'rF12';
	stDbReadQuery.stConfig.strStartTime[1] := '2026-03-04 15:21:32';
	stDbReadQuery.stConfig.strEndTime[1]   := '2026-03-04 15:21:32';

END_PROGRAM

PROGRAM _CYCLIC
	(* Insert code here *)

	guiDQHeartBeat;

END_PROGRAM

PROGRAM _EXIT
	(* Insert code here *)

END_PROGRAM
```

### Program Logical/DataSQLAla

#### Variables.var
```iecst
(*Alarm insert buffer + query - OPC ::DataSQLAla:*)
VAR
	AlarmInsertBuffer : AlarmInsertBuffer_typ;
	AlarmDataSQLQuery : DataSQLQuery_typ;
	UtcDTGetTime_0 : UtcDTGetTime;
	tonAlarm : TON;
	dtNow : DATE_AND_TIME;
	diAlarmCode : DINT;
	strTmp : STRING[16];
	bSimEnable : BOOL := TRUE;
END_VAR
```

#### Main.st
```iecst
PROGRAM _INIT
	AlarmDataSQLQuery.Config.PointName[0] := 'AlarmTime';
	AlarmDataSQLQuery.Config.PointName[1] := 'AlarmCode';
	AlarmDataSQLQuery.Config.PointName[2] := 'AlarmState';
	AlarmDataSQLQuery.Config.PointName[3] := 'AlarmText';
	bSimEnable := TRUE;
END_PROGRAM

PROGRAM _CYCLIC
	UtcDTGetTime_0.enable := TRUE;
	UtcDTGetTime_0();
	IF UtcDTGetTime_0.status = 0 THEN
		dtNow := UtcDTGetTime_0.DT1;
	END_IF

	(*随机报警插入：采集端 reset_trigger_after_read 清零后再次产生*)
	tonAlarm(IN := bSimEnable AND NOT AlarmInsertBuffer.InsertTrigger, PT := T#8s);
	IF EDGEPOS(tonAlarm.Q) THEN
		AlarmInsertBuffer.AlarmTime := dtNow;
		diAlarmCode := RandRange(1000, 1099);
		AlarmInsertBuffer.AlarmCode := DINT_TO_UDINT(diAlarmCode);
		AlarmInsertBuffer.AlarmState := DINT_TO_UDINT(RandRange(0, 1));
		strTmp := '';
		brsitoa(diAlarmCode, ADR(strTmp));
		AlarmInsertBuffer.AlarmText := 'SIM_ALARM_';
		brsstrcat(ADR(AlarmInsertBuffer.AlarmText), ADR(strTmp));
		AlarmInsertBuffer.AlarmBatch := gDataSQLBatch.BatchCode;
		AlarmInsertBuffer.InsertTrigger := TRUE;
	END_IF
END_PROGRAM

PROGRAM _EXIT

END_PROGRAM
```

### Program Logical/DataSQLAud

#### Variables.var
```iecst
(*Audit insert buffer + query - OPC ::DataSQLAud:*)
VAR
	AuditInsertBuffer : AuditInsertBuffer_typ;
	AuditDataSQLQuery : DataSQLQuery_typ;
	UtcDTGetTime_0 : UtcDTGetTime;
	tonAudit : TON;
	dtNow : DATE_AND_TIME;
	diAuditIdx : DINT;
	strTmp : STRING[16];
	bSimEnable : BOOL := TRUE;
END_VAR
```

#### Main.st
```iecst
PROGRAM _INIT
	AuditDataSQLQuery.Config.PointName[0] := 'AuditTime';
	AuditDataSQLQuery.Config.PointName[1] := 'AuditOperator';
	AuditDataSQLQuery.Config.PointName[2] := 'AuditText';
	bSimEnable := TRUE;
END_PROGRAM

PROGRAM _CYCLIC
	UtcDTGetTime_0.enable := TRUE;
	UtcDTGetTime_0();
	IF UtcDTGetTime_0.status = 0 THEN
		dtNow := UtcDTGetTime_0.DT1;
	END_IF

	(*随机审计插入：采集端 reset_trigger_after_read 清零后再次产生*)
	tonAudit(IN := bSimEnable AND NOT AuditInsertBuffer.InsertTrigger, PT := T#10s);
	IF EDGEPOS(tonAudit.Q) THEN
		AuditInsertBuffer.AuditTime := dtNow;
		diAuditIdx := RandRange(1, 9);
		strTmp := '';
		brsitoa(diAuditIdx, ADR(strTmp));
		AuditInsertBuffer.AuditOperator := 'Operator';
		brsstrcat(ADR(AuditInsertBuffer.AuditOperator), ADR(strTmp));
		AuditInsertBuffer.AuditText := 'SIM_AUDIT_EVENT_';
		brsstrcat(ADR(AuditInsertBuffer.AuditText), ADR(strTmp));
		AuditInsertBuffer.AuditBatch := gDataSQLBatch.BatchCode;
		AuditInsertBuffer.InsertTrigger := TRUE;
	END_IF
END_PROGRAM

PROGRAM _EXIT

END_PROGRAM
```

### Program Logical/DataSQLPro

#### Variables.var
```iecst
(*Product query config - OPC ::DataSQLPro:*)
VAR
	ProductDataSQLQuery : DataSQLQuery_typ;
END_VAR
```

#### Main.st
```iecst
PROGRAM _INIT
	ProductDataSQLQuery.Config.PointName[0] := 'DataProductTime';
	ProductDataSQLQuery.Config.PointName[1] := 'DataProductState';
	ProductDataSQLQuery.Config.PointName[2] := 'DataProductCH01';
	ProductDataSQLQuery.Config.PointName[3] := 'DataProductCH02';
	ProductDataSQLQuery.Config.PointName[4] := 'DataProductCH03';
	ProductDataSQLQuery.Config.PointName[5] := 'DataProductCH04';
	ProductDataSQLQuery.Config.PointName[6] := 'DataProductCH05';
	ProductDataSQLQuery.Config.PointName[7] := 'DataProductCH06';
END_PROGRAM

PROGRAM _CYCLIC
	(*查询配置由采集端/HMI写入，此处仅保持变量存在*)
	ProductDataSQLQuery;
END_PROGRAM

PROGRAM _EXIT

END_PROGRAM
```

### Program Logical/DataSQLRec

#### Variables.var
```iecst
(*Recipe query config - OPC ::DataSQLRec:*)
VAR
	RecipeDataSQLQuery : DataSQLQuery_typ;
END_VAR
```

#### Main.st
```iecst
PROGRAM _INIT
	RecipeDataSQLQuery.Config.PointName[0] := 'DataRecipeTime';
	RecipeDataSQLQuery.Config.PointName[1] := 'DataRecipeState';
	RecipeDataSQLQuery.Config.PointName[2] := 'DataRecipeCH00';
	RecipeDataSQLQuery.Config.PointName[3] := 'DataRecipeCH01';
	RecipeDataSQLQuery.Config.PointName[4] := 'DataRecipeCH02';
	RecipeDataSQLQuery.Config.PointName[5] := 'DataRecipeCH03';
	RecipeDataSQLQuery.Config.PointName[6] := 'DataRecipeCH04';
	RecipeDataSQLQuery.Config.PointName[7] := 'DataRecipeCH05';
	RecipeDataSQLQuery.Config.PointName[8] := 'DataRecipeCH06';
	RecipeDataSQLQuery.Config.PointName[9] := 'DataRecipeCH07';
	RecipeDataSQLQuery.Config.PointName[10] := 'DataRecipeCH08';
	RecipeDataSQLQuery.Config.PointName[11] := 'DataRecipeCH09';
	RecipeDataSQLQuery.Config.PointName[12] := 'DataRecipeCH10';
	RecipeDataSQLQuery.Config.PointName[13] := 'DataRecipeCH11';
	RecipeDataSQLQuery.Config.PointName[14] := 'DataRecipeCH12';
	RecipeDataSQLQuery.Config.PointName[15] := 'DataRecipeCH13';
	RecipeDataSQLQuery.Config.PointName[16] := 'DataRecipeCH14';
	RecipeDataSQLQuery.Config.PointName[17] := 'DataRecipeCH15';
	RecipeDataSQLQuery.Config.PointName[18] := 'DataRecipeCH16';
	RecipeDataSQLQuery.Config.PointName[19] := 'DataRecipeCH17';
	RecipeDataSQLQuery.Config.PointName[20] := 'DataRecipeCH18';
	RecipeDataSQLQuery.Config.PointName[21] := 'DataRecipeCH19';
	RecipeDataSQLQuery.Config.PointName[22] := 'DataRecipeCH20';
	RecipeDataSQLQuery.Config.PointName[23] := 'DataRecipeCH21';
	RecipeDataSQLQuery.Config.PointName[24] := 'DataRecipeCH22';
	RecipeDataSQLQuery.Config.PointName[25] := 'DataRecipeCH23';
	RecipeDataSQLQuery.Config.PointName[26] := 'DataRecipeCH24';
	RecipeDataSQLQuery.Config.PointName[27] := 'DataRecipeCH25';
END_PROGRAM

PROGRAM _CYCLIC
	(*查询配置由采集端/HMI写入，此处仅保持变量存在*)
	RecipeDataSQLQuery;
END_PROGRAM

PROGRAM _EXIT

END_PROGRAM
```

### Package Logical/LibAsHttp1_ST/HelloWorld - Simple Request Response Sample

### Program Logical/LibAsHttp1_ST/HelloWorld/client_1 (IEC) - Client Asking Ressource '/HelloWorld.cgi'

#### client_1.st - Implementation code
```iecst
(********************************************************************
 * COPYRIGHT -- Bernecker + Rainer
 ********************************************************************
 * Program: client_1
 * File: client_1.st
 * Author: Bernecker + Rainer
 * Created: February 16, 2012
 ********************************************************************
 * Implementation of program client_1
 ********************************************************************)

PROGRAM _INIT

	Ressource 				:= '/HelloWorld.cgi';

	Client.method 			:= httpMETHOD_GET;
	Client.option 			:= httpOPTION_HTTP_11;

	Client.pHost 			:= ADR(Host);
	Client.pUri 			:= ADR(Ressource);
	Client.pResponseData 	:= ADR(Responsedata);
	Client.responseDataSize := SIZEOF(Responsedata);

END_PROGRAM

PROGRAM _CYCLIC

	Client(enable := Doenable, send := Dosend); (* Call httpClient() *)

	(* TODO: Error handling *)

END_PROGRAM

PROGRAM _EXIT
	(* Release Client instance *)
	Client(enable := 0, send := 0);
END_PROGRAM
```

#### client_1.var - HTTP Client Variables
```iecst
(********************************************************************
 * COPYRIGHT --  Bernecker + Rainer
 ********************************************************************
 * Program: client_1
 * File: client_1.var
 * Author: Bernecker + Rainer
 * Created: February 16, 2012
 ********************************************************************
 * Local variables of program client_1
 ********************************************************************)
VAR
	Client : httpClient := (enable:=FALSE,send:=FALSE,abort:=FALSE,option:=0,pHost:=0,hostPort:=0,method:=httpMETHOD_GET,pUri:=0,pRequestHeader:=0,pRequestData:=0,requestDataLen:=0,pResponseHeader:=0,pResponseData:=0,responseDataSize:=0,pStatistics:=0,pStruct:=0,status:=0,tcpStatus:=0,httpStatus:=0,responseDataLen:=0,phase:=0,_i_state:=0,_i_result:=0,_ident:=0,_oldEnable:=0,_oldAbort:=0,_oldSend:=0,_state:=0,_internal:=0);
	Doenable : BOOL := FALSE; (*Enables FUB Instance*)
	Dosend : BOOL := FALSE; (*Sends request on positive edge*)
	Host : STRING[100] := 'localhost';
	Responsedata : STRING[80] := '';
	Ressource : STRING[80] := '';
END_VAR
```

### Program Logical/LibAsHttp1_ST/HelloWorld/service_1 (IEC) - Webservice 'HelloWorld.cgi'

#### service_1.st - Implementation code
```iecst
(********************************************************************
 * COPYRIGHT -- Bernecker + Rainer
 ********************************************************************
 * Program: service_1
 * File: service_1.st
 * Author: Bernecker + Rainer
 * Created: February 16, 2012
 ********************************************************************
 * Implementation of program service_1
 ********************************************************************)

PROGRAM _INIT

	Webservice.pServiceName 	:= ADR('helloworld.cgi'); (* Name of webservice *)
	Webservice.option 			:= httpOPTION_HTTP_10 + httpOPTION_SERVICE_TYPE_NAME;

	Response 					:= 'Hello client';
	Webservice.pResponseData 	:= ADR(Response);
	Webservice.responseDataLen 	:= strlen(ADR(Response));

	(* Register Webservice*)
	Webservice(enable := 1);

END_PROGRAM

PROGRAM _CYCLIC

	IF  Webservice.send = TRUE  THEN
		Webservice.send := FALSE; (* Reset *)
	ELSIF Webservice.status = ERR_OK AND Webservice.send = FALSE THEN
		(* Create Response *)
		Webservice.responseDataLen := strlen(ADR(Response));
		Webservice.send := TRUE; (* Send on positive edge*)
	END_IF

	Webservice();
END_PROGRAM

PROGRAM _EXIT

	(* Unregister Webservice *)
	Webservice(enable := 0);

END_PROGRAM
```

#### service_1.var - HTTP Service Variables
```iecst
(********************************************************************
 * COPYRIGHT --  Bernecker + Rainer
 ********************************************************************
 * Program: service_1
 * File: service_1.var
 * Author: Bernecker + Rainer
 * Created: February 16, 2012
 ********************************************************************
 * Local variables of program service_1
 ********************************************************************)
VAR
	Response : STRING[80] := '';
	Webservice : httpService := (0);
END_VAR
```

### Package Logical/LibAsHttp1_ST/Counter - Dynamic Response Data Sample

### Program Logical/LibAsHttp1_ST/Counter/client_2 (IEC) - Client Asking Ressource '/Counter.cgi'

#### client_2.st - Implementation code
```iecst
(********************************************************************
 * COPYRIGHT -- Bernecker + Rainer
 ********************************************************************
 * Program: Client_2
 * File: Client_2.st
 * Author: Bernecker + Rainer
 * Created: February 17, 2012
 ********************************************************************
 * Implementation of program Client_2
 ********************************************************************)
PROGRAM _INIT

	Ressource 				:= '/Counter.cgi';	(* Name of file or webservice to be requested *)
	Client.pUri 			:= ADR(Ressource);
	Client.method 			:= httpMETHOD_GET; 	(* Request method *)

	Client.option 			:= httpOPTION_HTTP_11;
	Client.pHost 			:= ADR(Host); 		(* Host to connect to *)

	Client.pResponseData 	:= ADR(Responsedata);
	Client.responseDataSize := SIZEOF(Responsedata);

END_PROGRAM

PROGRAM _CYCLIC

	Client(enable := Doenable, send := Dosend); (* Call httpClient() *)

	(* TODO: Error handling *)

END_PROGRAM

PROGRAM _EXIT

	(* Release Client instance *)
	Client(enable := 0, send := 0);

END_PROGRAM
```

#### client_2.var - HTTP Client Variables
```iecst
(********************************************************************
 * COPYRIGHT --  Bernecker + Rainer
 ********************************************************************
 * Program: Client_2
 * File: Client_2.var
 * Author: Bernecker + Rainer
 * Created: February 17, 2012
 ********************************************************************
 * Local variables of program Client_2
 ********************************************************************)
VAR
	Client : httpClient := (enable:=FALSE,send:=FALSE,abort:=FALSE,option:=0,pHost:=0,hostPort:=0,method:=httpMETHOD_GET,pUri:=0,pRequestHeader:=0,pRequestData:=0,requestDataLen:=0,pResponseHeader:=0,pResponseData:=0,responseDataSize:=0,pStatistics:=0,pStruct:=0,status:=0,tcpStatus:=0,httpStatus:=0,responseDataLen:=0,phase:=0,_i_state:=0,_i_result:=0,_ident:=0,_oldEnable:=0,_oldAbort:=0,_oldSend:=0,_state:=0,_internal:=0); (*httpClient instance*)
	Doenable : BOOL := FALSE; (*Enables FUB Instance*)
	Dosend : BOOL := FALSE; (*Sends request on positive edge*)
	Host : STRING[100] := 'localhost'; (*Server to connect to*)
	Responsedata : STRING[80] := ''; (*buffer for response data*)
	Ressource : STRING[80] := ''; (*file or webservice to be requested*)
END_VAR
```

### Program Logical/LibAsHttp1_ST/Counter/service_2 (IEC) - Webservice 'Counter.cgi'

#### service_2.st - Implementation code
```iecst
(********************************************************************
 * COPYRIGHT -- Bernecker + Rainer
 ********************************************************************
 * Program: service_2
 * File: service_2.st
 * Author: Bernecker + Rainer
 * Created: February 17, 2012
 ********************************************************************
 * Implementation of program service_2
 ********************************************************************)

PROGRAM _INIT

	Webservice.pServiceName 	:= ADR('Counter.cgi'); (* Name of webservice *)
	Webservice.option 			:= httpOPTION_HTTP_10 + httpOPTION_SERVICE_TYPE_NAME;

	Webservice.pResponseData 	:= ADR(Response);
	Webservice.pResponseHeader  := ADR(ResponseHeader);

	(* Register Webservice*)
	Webservice(enable := 1);
END_PROGRAM

PROGRAM _CYCLIC

	IF  Webservice.send = TRUE  THEN
		Webservice.send := FALSE; (* Reset *)
	ELSIF Webservice.status = ERR_OK AND Webservice.phase = httpPHASE_RECEIVED AND Webservice.send = FALSE THEN
		(* Create Response *)
		ResponseHeader.contentType 	:= 'text/plain'; (* Response is plain text data and this is the correct MIME type *)

		Helper 						:= (UINT_TO_STRING(Counter));
		Counter 					:= Counter + 1;
		Response 					:= 'This webservice was requested ';
		strcat(ADR(Response), ADR(Helper));
		strcat(ADR(Response), ADR(' times.'));

		Webservice.responseDataLen 	:= strlen(ADR(Response)); (* Length of the response *)
		Webservice.send 			:= TRUE; (* Send on positive edge*)
	END_IF

	Webservice();
END_PROGRAM

PROGRAM _EXIT

	(* Unregister Webservice *)
	Webservice(enable := 0);

END_PROGRAM
```

#### service_2.var - HTTP Service Variables
```iecst
(********************************************************************
 * COPYRIGHT --  Bernecker + Rainer
 ********************************************************************
 * Program: service_2
 * File: service_2.var
 * Author: Bernecker + Rainer
 * Created: February 17, 2012
 ********************************************************************
 * Local variables of program service_2
 ********************************************************************)
VAR
	Counter : UINT := 0;
	Helper : STRING[10];
	Response : STRING[80] := '';
	ResponseHeader : httpResponseHeader_t := (0);
	Webservice : httpService := (0);
END_VAR
```

### Package Logical/LibAsHttp1_ST/Proxy - Communication Via Proxy (HTTP Communication Inspection)

### Program Logical/LibAsHttp1_ST/Proxy/client_3 (IEC) - Client Asking Ressource '/Proxy.cgi' Via A Local Proxy (Port 8888)

#### client_3.st - Implementation code
```iecst
(********************************************************************
 * COPYRIGHT -- Bernecker + Rainer
 ********************************************************************
 * Program: Client_2
 * File: Client_2.st
 * Author: Bernecker + Rainer
 * Created: February 17, 2012
 ********************************************************************
 * Implementation of program Client_2
 ********************************************************************)

PROGRAM _INIT
	(* Fiddler is a HTTP Proxy for HTTP diagnostics http://www.fiddler2.com/fiddler2/ *)

	(* Proxy specific *)
	Client.pHost 			:= ADR(Proxy); 		(* Host to connect to: Proxy*)
	Client.hostPort 		:= Proxyport;  		(* Port of the proxy *)

	Requestheader.host 		:= Host;			(* Required field in HTTP/1.1. Normally generated
													automaticly using "Client.pHost". When a proxy
													is used, this field should be set explictly. *)
	Client.pRequestHeader 	:= ADR(Requestheader);

	Ressource				:= 'http://'; 		(* Communication over a proxy requires full request path. *)
	strcat(ADR(Ressource), ADR(Host));
	(* Not proxy specific *)
	strcat(ADR(Ressource), ADR('/Proxy.cgi'));	(* Name of file or webservice to be requested *)
	Client.pUri 			:= ADR(Ressource);
	Client.method 			:= httpMETHOD_GET;	(* Request method *)
	Client.option 			:= httpOPTION_HTTP_11;

	Client.pResponseData 	:= ADR(Responsedata);
	Client.responseDataSize := SIZEOF(Responsedata);

END_PROGRAM

PROGRAM _CYCLIC

	IF Doenable = FALSE THEN
		_Connectioninformation 	:= 'FUB disabled';
		Client.pHost 			:= ADR(Proxy); 		(* Host to connect to: Proxy*)
		Client.hostPort 		:= Proxyport;  		(* Port of the proxy *)

		Requestheader.host 		:= Host;			(* Required field in HTTP/1.1. Normally generated
													automaticly using "Client.pHost". When a proxy
													is used, this field should be set explictly. *)

	ELSIF Dosend = FALSE THEN
		_Connectioninformation 	:= 'Dosend set to false';  	 	(* Reset message *)
	ELSIF Client.status = httpERR_CLIENT_TCP_INVALID_HOST OR Client.status = httpERR_CLIENT_TCP_CONN_FAILED THEN
		(* Check proxy configuration and availability *)
		_Connectioninformation 	:= 'Could not connect: Check proxy configuration and availability';
	ELSIF Client.status = ERR_OK OR Client.status = httpERR_CLIENT_TCP_CONN_CLOSED THEN
		_Connectioninformation 	:= '';  				(* Reset message *)
	END_IF

	mylen := strlen(ADR(Responsedata));

	Client(enable := Doenable, send := Dosend); 	(* Call httpClient() *)
	(* TODO: Error handling *)
END_PROGRAM

PROGRAM _EXIT
	Client(enable := 0, send := 0);			(* Release Client instance *)
END_PROGRAM
```

#### client_3.var - HTTP Client Variables
```iecst
(********************************************************************
 * COPYRIGHT --  Bernecker + Rainer
 ********************************************************************
 * Program: Client_2
 * File: Client_2.var
 * Author: Bernecker + Rainer
 * Created: February 17, 2012
 ********************************************************************
 * Local variables of program Client_2
 ********************************************************************)
VAR
	mylen : UDINT := 0;
	_Connectioninformation : STRING[80] := '';
	Client : httpClient; (*httpClient instance*)
	Doenable : BOOL := FALSE; (*Enables FUB Instance*)
	Dosend : BOOL := FALSE; (*Sends request on positive edge*)
	Host : STRING[100] := 'localhost:80'; (*Webserver and Port  to connect to*)
	Proxy : STRING[100] := '127.0.0.1'; (*Proxy to connect to*)
	Proxyport : UINT := 8888; (*Port of proxy*)
	Requestheader : httpRequestHeader_t := (0);
	Responsedata : STRING[300]; (*buffer for response data*)
	Ressource : STRING[80] := ''; (*file or webservice to be requested*)
END_VAR
```

### Program Logical/LibAsHttp1_ST/Proxy/service_3 (IEC) - Webservice 'Formdata.cgi'

#### service_3.st - Implementation code
```iecst
(********************************************************************
 * COPYRIGHT -- Bernecker + Rainer
 ********************************************************************
 * Program: service_3
 * File: service_3.st
 * Author: Bernecker + Rainer
 * Created: February 17, 2012
 ********************************************************************
 * Implementation of program service_3
 ********************************************************************)

PROGRAM _INIT

	Webservice.pServiceName 			:= ADR('Proxy.cgi'); (* Name of webservice *)
	Webservice.option 					:= httpOPTION_HTTP_10 + httpOPTION_SERVICE_TYPE_NAME;

	Webservice.pResponseData 			:= ADR(Response);

	Webservice.pRequestHeader 			:= ADR(RequestHeader);
	RequestHeader.rawHeader.pData 		:= ADR(RequestRawHeader);
	RequestHeader.rawHeader.dataSize 	:= SIZEOF(RequestRawHeader);

	(* Register Webservice*)
	Webservice(enable := 1);
END_PROGRAM

PROGRAM _CYCLIC

	IF (Webservice.send = TRUE) THEN
		Webservice.send := FALSE; (* Reset *)
	ELSIF (Webservice.status = ERR_OK) AND (Webservice.send = FALSE) THEN
		(* Create Response *)
		strcpy(ADR(Response) , ADR('Some Data.'));
		Webservice.responseDataLen := strlen(ADR(Response)); (* Length of the response *)
		Webservice.send := TRUE; (* Send on positive edge*)
	END_IF

	Webservice();
END_PROGRAM

PROGRAM _EXIT

	(* Unregister Webservice *)
	Webservice(enable := 0);

END_PROGRAM
```

#### service_3.var - HTTP Service Variables
```iecst
(********************************************************************
 * COPYRIGHT --  Bernecker + Rainer
 ********************************************************************
 * Program: service_3
 * File: service_3.var
 * Author: Bernecker + Rainer
 * Created: February 17, 2012
 ********************************************************************
 * Local variables of program service_3
 ********************************************************************)
VAR
	Webservice : httpService := (0);
	RequestHeader : httpRequestHeader_t := (0);
	Response : STRING[300];
	RequestRawHeader : STRING[200] := '';
END_VAR
```

### Package Logical/LibAsHttp1_ST/FormularData - Simple Form Sample

### Program Logical/LibAsHttp1_ST/FormularData/client_4 (IEC) - Client Sends 2 Parameter

#### client_4.st - Implementation code
```iecst
(********************************************************************
 * COPYRIGHT -- Bernecker + Rainer
 ********************************************************************
 * Program: client_4
 * File: client_4.st
 * Author: Bernecker + Rainer
 * Created: February 16, 2012
 ********************************************************************
 * Implementation of program client_4
 ********************************************************************)

PROGRAM _INIT

	Ressource 				:= '/formdata.cgi';

	Client.method 			:= httpMETHOD_POST;
	Client.option 			:= httpOPTION_HTTP_11;

	Client.pHost 			:= ADR(Host);
	Client.pUri 			:= ADR(Ressource);
	Client.pResponseData 	:= ADR(Responsedata);
	Client.responseDataSize := SIZEOF(Responsedata);
	Client.pRequestData		:= ADR(Request);

END_PROGRAM

PROGRAM _CYCLIC

	IF Dosend = FALSE AND Doenable = TRUE THEN
		SetParam.enable := TRUE;
		Request 		:= '';
		SetParam.pDest 	:= ADR(Request);
		SetParam.destSize := SIZEOF(Request);
		SetParam.pParam := ADR('usertext1');
		SetParam.pValue := ADR(userText1);
		SetParam();

		SetParam.pParam := ADR('usertext2');
		SetParam.pValue := ADR(userText2);
		SetParam();
		Client.requestDataLen := SetParam.destLen;
	END_IF

	Client(enable := Doenable, send := Dosend); (* Call httpClient() *)

	(* TODO: Error handling *)

END_PROGRAM

PROGRAM _EXIT
	(* Release Client instance *)
	Client(enable := 0, send := 0);
END_PROGRAM
```

#### client_4.var - HTTP Client Variables
```iecst
(********************************************************************
 * COPYRIGHT --  Bernecker + Rainer
 ********************************************************************
 * Program: client_4
 * File: client_4.var
 * Author: Bernecker + Rainer
 * Created: February 16, 2012
 ********************************************************************
 * Local variables of program client_4
 ********************************************************************)
VAR
	Client : httpClient := (enable:=FALSE,send:=FALSE,abort:=FALSE,option:=0,pHost:=0,hostPort:=0,method:=httpMETHOD_GET,pUri:=0,pRequestHeader:=0,pRequestData:=0,requestDataLen:=0,pResponseHeader:=0,pResponseData:=0,responseDataSize:=0,pStatistics:=0,pStruct:=0,status:=0,tcpStatus:=0,httpStatus:=0,responseDataLen:=0,phase:=0,_i_state:=0,_i_result:=0,_ident:=0,_oldEnable:=0,_oldAbort:=0,_oldSend:=0,_state:=0,_internal:=0);
	Doenable : BOOL := FALSE; (*Enables FUB Instance*)
	Dosend : BOOL := FALSE; (*Sends request on positive edge*)
	Host : STRING[100] := 'localhost';
	Request : STRING[200];
	Responsedata : ARRAY[0..4] OF STRING[80];
	Ressource : STRING[80] := '';
	userText1 : STRING[80] := '';
	userText2 : STRING[80] := '';
	SetParam : httpSetParamUrl := (0);
END_VAR
```

### Program Logical/LibAsHttp1_ST/FormularData/service_4 (IEC) - Webservice Evaluates Form Data

#### service_4.st - Implementation code
```iecst
(********************************************************************
 * COPYRIGHT -- Bernecker + Rainer
 ********************************************************************
 * Program: service_4
 * File: service_4.st
 * Author: Bernecker + Rainer
 * Created: February 16, 2012
 ********************************************************************
 * Implementation of program service_4
 ********************************************************************)

PROGRAM _INIT

	Webservice.pServiceName 	:= ADR('formdata.cgi'); (* Name of webservice *)
	Webservice.option 			:= httpOPTION_HTTP_11 + httpOPTION_SERVICE_TYPE_NAME;
	Webservice.pResponseHeader  := ADR(ResponseHeader);
	Webservice.pRequestData  	:= ADR(Request);
	Webservice.requestDataSize  := SIZEOF(Request);
	Webservice.pResponseData 	:= ADR(Response);

	(* Register Webservice*)
	Webservice(enable := 1);

END_PROGRAM

PROGRAM _CYCLIC

	IF  Webservice.send = TRUE  THEN
		Webservice.send := FALSE; (* Reset *)
	ELSIF Webservice.status = ERR_OK AND Webservice.send = FALSE AND Webservice.phase = httpPHASE_RECEIVED THEN
		(* Create Response *)
		ResponseHeader.contentType 	:= 'text/html'; (* Response is HTML data and this is the correct MIME type *)
		IF Webservice.method = httpMETHOD_POST THEN

			UrlParam.enable := TRUE;
			UrlParam.pParam := ADR('usertext1');
			UrlParam.pSrc := ADR(Request);
			UrlParam.pValue := ADR(FormParam1);
			UrlParam.valueSize := SIZEOF(FormParam1);
			UrlParam();
			strcpy( strcpy( strcpy(ADR(Response) , ADR('<html><body><h2>Form Result</h2><p>First field contained: <i>')), ADR(FormParam1)), ADR('</i></p>') ) ;

			UrlParam.pParam := ADR('usertext2');
			UrlParam.pValue := ADR(FormParam2);
			UrlParam.valueSize := SIZEOF(FormParam2);
			UrlParam();
			strcat(ADR(Response),ADR('<p>Second field contained: <i>'));
			strcat(ADR(Response), ADR(FormParam2));
			strcat(ADR(Response),ADR('</i></p></body></html>'));
		ELSE
			Response := '<html><body><h2>Simple Form</h2><form method="POST" action="/formdata.cgi"><input type="text" name="usertext1" size="20" /><br><input type="text" name="usertext2" size="20" /><br><input type="submit" name="bt1" value="Submit"></form></body></html>';
		END_IF

		Webservice.responseDataLen := strlen(ADR(Response));
		Webservice.send := TRUE; (* Send on positive edge*)
	END_IF

	Webservice();
END_PROGRAM

PROGRAM _EXIT

	(* Unregister Webservice *)
	Webservice(enable := 0);

END_PROGRAM
```

#### service_4.var - HTTP Service Variables
```iecst
(********************************************************************
 * COPYRIGHT --  Bernecker + Rainer
 ********************************************************************
 * Program: service_4
 * File: service_4.var
 * Author: Bernecker + Rainer
 * Created: February 16, 2012
 ********************************************************************
 * Local variables of program service_4
 ********************************************************************)
VAR
	Request : STRING[400];
	ResponseHeader : httpResponseHeader_t := (0);
	Response : STRING[400];
	Webservice : httpService := (0);
	UrlParam : httpGetParamUrl := (0);
	FormParam1 : STRING[80] := '';
	FormParam2 : STRING[80] := '';
END_VAR
```

### Program Logical/ParallelTest

#### Variables.var
```iecst
VAR
	usiTestModel : USINT;
	usiIdx : USINT;
END_VAR
(*Insert your comment here.*)
VAR
	bExecuteRead : BOOL;
	stDbReadQuery : dbReadQuery_typ;
	bParallelTriger : ARRAY[0..MY_DATA_SIZE_MINUS_ONE] OF BOOL;
	uiHeartBeat : UINT;
	uiQueryFeedBack : UINT;
END_VAR
(*DATA POINT*)
VAR
	F1 : ARRAY[0..MY_DATA_SIZE_MINUS_ONE] OF REAL;
	F2 : ARRAY[0..MY_DATA_SIZE_MINUS_ONE] OF REAL;
	F3 : ARRAY[0..MY_DATA_SIZE_MINUS_ONE] OF REAL;
	F4 : ARRAY[0..MY_DATA_SIZE_MINUS_ONE] OF REAL;
	F5 : ARRAY[0..MY_DATA_SIZE_MINUS_ONE] OF REAL;
END_VAR
(*CONSTANT*)
VAR CONSTANT
	MY_DATA_SIZE : UDINT := 100;
	MY_DATA_SIZE_MINUS_ONE : UDINT := MY_DATA_SIZE-1;
END_VAR
```

#### Main.st
```iecst
PROGRAM _INIT
	(* Insert code here *)

END_PROGRAM

PROGRAM _CYCLIC
	(* Insert code here *)
	IF usiTestModel = 10 THEN
		usiTestModel := 0;

		usiIdx := 0;
		bParallelTriger[usiIdx] := TRUE;
		F1[usiIdx] := usiIdx + 1;
		F2[usiIdx] := usiIdx + 2;
		F3[usiIdx] := usiIdx + 3;
		F4[usiIdx] := usiIdx + 4;
		F5[usiIdx] := usiIdx + 5;

		usiIdx := 10;
		bParallelTriger[usiIdx] := TRUE;
		F1[usiIdx] := usiIdx + 1;
		F2[usiIdx] := usiIdx + 2;
		F3[usiIdx] := usiIdx + 3;
		F4[usiIdx] := usiIdx + 4;
		F5[usiIdx] := usiIdx + 5;

		usiIdx := 49;
		bParallelTriger[usiIdx] := TRUE;
		F1[usiIdx] := usiIdx + 1;
		F2[usiIdx] := usiIdx + 2;
		F3[usiIdx] := usiIdx + 3;
		F4[usiIdx] := usiIdx + 4;
		F5[usiIdx] := usiIdx + 5;
	END_IF

END_PROGRAM

PROGRAM _EXIT
	(* Insert code here *)

END_PROGRAM
```

### Program Logical/pulldata (IEC)

#### Main.st - Init, cyclic, exit code
```iecst
(******************************************************************************
 * B&R AsHttp Library - POST JSON Data Example
 * Description: Send PLC data to HTTP server in JSON format
 * Library: AsHttp
 ******************************************************************************)

PROGRAM _INIT

    (* Initialize HTTP client *)
	httpClient_0.enable := TRUE;
	httpClient_0.pHost := ADR('127.0.0.1');  (* Server IP address *)
	httpClient_0.hostPort := 8000;               (* Server port *)

	(* Initialize state machine *)
	step := 0;
	sendTimer := 0;
	dataIndex := 0;

END_PROGRAM

PROGRAM _CYCLIC

	CASE step OF

		(* Step 0: Wait and prepare data *)
		0:
			sendTimer := sendTimer + 1;
			IF sendTimer >= 500 THEN  (* Send every 500ms (assuming 1ms cycle) *)
				sendTimer := 0;

				(* Get PLC variable value *)
				brsmemcpy(ADR(currentValue),ADR(PLCVariable),SIZEOF(PLCVariable));

				(* Build JSON string *)
				(* Format: [[timestamp1, value1], [timestamp2, value2], ...] *)

				(* For single point: *)
				jsonLength := BuildSinglePointJSON(
				ADR(jsonBuffer),
				SIZEOF(jsonBuffer),
				currentTimestamp,
				currentValue
				);

				step := 1;
			END_IF

			(* Step 1: Send POST request *)
		1:
			httpClient_0.send := TRUE;
			httpClient_0.pUri := ADR('/api/data');
			httpClient_0.pRequestHeader := ADR(requestHeader);
			httpClient_0.pRequestData := ADR(jsonBuffer);
			httpClient_0.requestDataLen := jsonLength;
			httpClient_0.httpMethod := httpMETHOD_POST;

			IF httpClient_0.status = 0 THEN
				step := 2;
			ELSIF httpClient_0.status < 0 THEN
				(* Error handling *)
				errorCode := httpClient_0.status;
				step := 10;
			END_IF

			(* Step 2: Wait for response *)
		2:
			httpClient_0.send := FALSE;

			IF httpClient_0.responseDataLen > 0 THEN
				(* Response received *)
				responseCode := httpClient_0.responseCode;
				step := 0;
			ELSIF httpClient_0.status < 0 THEN
				errorCode := httpClient_0.status;
				step := 10;
			END_IF

			(* Step 10: Error state *)
		10:
			(* Wait and retry *)
			sendTimer := sendTimer + 1;
			IF sendTimer >= 5000 THEN
				sendTimer := 0;
				step := 0;
			END_IF

	END_CASE

	(* Call HTTP client function block *)
	httpClient_0();

END_PROGRAM
```

#### Types.typ - Local data types
```iecst
TYPE
	data_typ : 	STRUCT
		value : REAL;
		ts : UDINT;
	END_STRUCT;
END_TYPE
```

#### Variables.var - Local variables
```iecst
(* HTTP Client *)
VAR
	httpClient_0 : httpClient; (* Request/Response buffers *)
	jsonBuffer : ARRAY[0..8191] OF USINT;
	jsonLength : UDINT;
	responseBuffer : ARRAY[0..4095] OF USINT; (* Request header - Content-Type: application/json *)
	requestHeader : STRING[256] := 'Content-Type: application/json'; (* State machine *)
	step : UINT;
	sendTimer : UDINT;
	errorCode : DINT;
	responseCode : UINT; (* Data *)
	currentTimestamp : UDINT;
	currentValue : ARRAY[0..3599] OF data_typ;
	PLCVariable : ARRAY[0..3599] OF data_typ; (* Batch data storage (for 3600 points) *)
	DTGetTime_0 : DTGetTime;
END_VAR
```

#### Ref.st - Init, cyclic, exit code
```iecst
(******************************************************************************
 * B&R AsHttp Library - POST JSON Data Example
 * Description: Send PLC data to HTTP server in JSON format
 * Library: AsHttp
 ******************************************************************************)

PROGRAM _INIT

    (* Initialize HTTP client *)
	httpClient_0.enable := TRUE;
	httpClient_0.pHost := ADR('127.0.0.1');  (* Server IP address *)
	httpClient_0.hostPort := 8000;               (* Server port *)

	(* Initialize state machine *)
	step := 0;
	sendTimer := 0;
	dataIndex := 0;

END_PROGRAM

PROGRAM _CYCLIC

    (* Call HTTP client function block *)
	httpClient(httpClient_0);

	CASE step OF

		(* Step 0: Wait and prepare data *)
		0:
			sendTimer := sendTimer + 1;
			IF sendTimer >= 500 THEN  (* Send every 500ms (assuming 1ms cycle) *)
				sendTimer := 0;

				(* Get current timestamp (Unix format) *)
				currentTimestamp := GetUnixTimestamp();

				(* Get PLC variable value *)
				currentValue := PLCVariable;

				(* Build JSON string *)
				(* Format: [[timestamp1, value1], [timestamp2, value2], ...] *)

				(* For single point: *)
				jsonLength := BuildSinglePointJSON(
				ADR(jsonBuffer),
				SIZEOF(jsonBuffer),
				currentTimestamp,
				currentValue
				);

				step := 1;
			END_IF

			(* Step 1: Send POST request *)
		1:
			httpClient_0.send := TRUE;
			httpClient_0.pUri := ADR('/api/data');
			httpClient_0.pRequestHeader := ADR(requestHeader);
			httpClient_0.pRequestData := ADR(jsonBuffer);
			httpClient_0.requestDataLen := jsonLength;
			httpClient_0.httpMethod := httpMETHOD_POST;

			IF httpClient_0.status = 0 THEN
				step := 2;
			ELSIF httpClient_0.status < 0 THEN
				(* Error handling *)
				errorCode := httpClient_0.status;
				step := 10;
			END_IF

			(* Step 2: Wait for response *)
		2:
			httpClient_0.send := FALSE;

			IF httpClient_0.responseDataLen > 0 THEN
				(* Response received *)
				responseCode := httpClient_0.responseCode;
				step := 0;
			ELSIF httpClient_0.status < 0 THEN
				errorCode := httpClient_0.status;
				step := 10;
			END_IF

			(* Step 10: Error state *)
		10:
			(* Wait and retry *)
			sendTimer := sendTimer + 1;
			IF sendTimer >= 5000 THEN
				sendTimer := 0;
				step := 0;
			END_IF

	END_CASE

END_PROGRAM
```

#### BuildJson.st
```iecst
ACTION Action:

END_ACTION
```

### Program Logical/TimeSt

#### Variables.var
```iecst
(*Insert your comment here.*)
VAR
	stRTCtime : RTCtime_typ;
	sDbDateTime : STRING[32];
END_VAR
```

#### Main.c
```c
#include <bur/plctypes.h>
#include <AsBrStr.h>

#ifdef _DEFAULT_INCLUDES
	#include <AsDefault.h>
#endif

static void append_usint_2d(char *dest, USINT v)
{
	char t[8];

	if (v < 10U)
		brsstrcat((UDINT)(unsigned long)dest, (UDINT)(unsigned long)"0");
	brsitoa((DINT)(UINT)v, (UDINT)(unsigned long)t);
	brsstrcat((UDINT)(unsigned long)dest, (UDINT)(unsigned long)t);
}

static void RTCtime_to_db_datetime_string(const RTCtime_typ *rtc, char *dest, UINT destSize)
{
	char ybuf[16];
	UINT y;

	if (destSize == 0U)
		return;

	brsmemset((UDINT)(unsigned long)dest, 0, (UDINT)destSize);

	y = rtc->year;
	if (y < 1000U)
		y += 1984U;

	brsitoa((DINT)y, (UDINT)(unsigned long)ybuf);
	brsstrcpy((UDINT)(unsigned long)dest, (UDINT)(unsigned long)ybuf);
	brsstrcat((UDINT)(unsigned long)dest, (UDINT)(unsigned long)"-");
	append_usint_2d(dest, rtc->month);
	brsstrcat((UDINT)(unsigned long)dest, (UDINT)(unsigned long)"-");
	append_usint_2d(dest, rtc->day);
	brsstrcat((UDINT)(unsigned long)dest, (UDINT)(unsigned long)" ");
	append_usint_2d(dest, rtc->hour);
	brsstrcat((UDINT)(unsigned long)dest, (UDINT)(unsigned long)":");
	append_usint_2d(dest, rtc->minute);
	brsstrcat((UDINT)(unsigned long)dest, (UDINT)(unsigned long)":");
	append_usint_2d(dest, rtc->second);
}

void _INIT ProgramInit(void)
{

}

void _CYCLIC ProgramCyclic(void)
{
	RTC_gettime(&stRTCtime);
	RTCtime_to_db_datetime_string(&stRTCtime, (char *)sDbDateTime, (UINT)sizeof(sDbDateTime));
}

void _EXIT ProgramExit(void)
{

}
```

### Program Logical/Trend

#### Variables.var
```iecst
(*DATA BASE Query*)
VAR
	stDbReadQuery : dbReadQuery_typ;
	bExecuteRead : BOOL;
END_VAR
(*DATA BASE CONSTANT*)
VAR CONSTANT
	REV_BUFFER_SIZE : UINT := 10000;
	REV_BUFFER_SIZE_MINUS_ONE : UINT := REV_BUFFER_SIZE-1;
	DB_READ_QUERY_SIZE : UINT := 10;
	DB_READ_QUERY_SIZE_MINUS_ONE : UINT := DB_READ_QUERY_SIZE-1;
END_VAR
(*Insert your comment here.*)
VAR CONSTANT
	MAX_ENTRIES_PERPAGE_MINUSONE : UINT := MAX_ENTRIES_PERPAGE- 1;
	MAX_ENTRIES_PERPAGE : UINT := 15;
END_VAR
VAR
	Trenddata : DINT;
END_VAR
```

#### Main.st
```iecst
PROGRAM _INIT
	(* Insert code here *)

END_PROGRAM

PROGRAM _CYCLIC
	(* Insert code here *)
		//Data GEN
	Trenddata:= RandRange(1,10);

	stDbReadQuery;
	bExecuteRead;

END_PROGRAM

PROGRAM _EXIT
	(* Insert code here *)

END_PROGRAM
```

Listed in the project but not available here: Logical/Libraries/BrRand/BrRand.typ, Logical/Libraries/BrRand/BrRand.var, Logical/Archive/AlarmQuerry/Types.typ, Logical/Archive/AuditQuerry, Logical/Archive/TimeSt, Logical/SMA/DataSQLBat/Types.typ
